REGION Network 1: Block description — Sections 1 to 3
   // ▀▀▀▀▀▀▀▀▀▀▀▀▀▀▀▀▀▀▀▀▀▀▀▀▀▀▀▀▀▀▀▀▀▀▀▀▀▀▀▀▀▀▀▀
   // 
   // TITLE:    STANDARD SYSTEM GLOBAL DATA
   // 
   // ▄▄▄▄▄▄▄▄▄▄▄▄▄▄▄▄▄▄▄▄▄▄▄▄▄▄▄▄▄▄▄▄▄▄▄▄▄▄▄▄▄▄▄▄
   //  
   // 
   // 
   // This is an essential system block that generates the internal logic and timing signals needed by 
   // all the other PAL software modules.
   // 
   // The block records the controller scan times and converts the Controller real time clock value 
   // to discrete integers, making the data globally available to all systems including non-Siemens 
   // equipment.
   // 
   // The block provides the following functions:
   // 
   //    •   Generates global logic signals (TRUE and FALSE)
   // 
   //    •   Generates the following scan synchronised timing pulses:
   //      50ms, 100ms, 200ms, 500ms, 1s and 2s
   // 
   //    •   Generates the following (1:1 mark/space) square wave signals:
   //      100ms, 200ms, 500ms, 1s and 2s
   // 
   //    •   Generates odd and even (alternating) cycle tick-tock signals
   // 
   //    •   Generates a first-cycle signal indicating the controller has just started
   // 
   //    •   Records the cycle time of the last, maximum and minimum controller cycles
   // 
   //    •   Reads the controller internal real time clock and converts the values to discrete 
   //      integer values containing: year, month, day, day of week, hour, minute, second 
   //      and millisecond
   // 
   // The block requires that the controller clock memory function is enabled.
   // 
   // The block must be the first non-debug block call within the main organisation block (OB 1).
   // 
   // 
   // 
   // 
   // 
   // ▄▄▄▄▄▄▄▄▄▄▄▄▄▄▄▄▄▄▄▄▄▄▄▄▄▄▄▄▄▄▄▄▄▄▄▄▄▄▄▄▄▄▄▄
   // 1.     BLOCK TECHNICAL SUMMARY
   // 
   // 
   //  ――――――――――――――――――――――――――――――――――――――――――
   //  NOMENCLATURE & ADDRESSING
   //  ――――――――――――――――――――――――――――――――――――――――――
   //  BLOCK TITLE         Standard System Global Data
   //  BLOCK FUNCTION GROUP    System
   //  BLOCK ADDRESS       FC 01001
   //  BLOCK SYMBOL        FC01001_StdSysGlobalData
   //  BLOCK USER ID         StdSysGlobalData
   // 
   //  ――――――――――――――――――――――――――――――――――――――――――
   //  BLOCK TYPE & USAGE
   //  ――――――――――――――――――――――――――――――――――――――――――
   //  BLOCK TYPE         Function (FC)
   //  BLOCK NUMBER        01001
   //  LANGUAGE           LAD
   //  OPTIMISED ACCESS     Yes
   //  PAL USAGE TYPE       Standard block
   // 
   //  ――――――――――――――――――――――――――――――――――――――――――
   //  METRICS
   //  ――――――――――――――――――――――――――――――――――――――――――
   //  LANGUAGE           LAD
   //  EXECUTION TIME       240.20 μs¹
   //  LOAD MEMORY         43.40 kB  (44440 bytes)
   //  WORK MEMORY             1.29 kB    (1322 bytes)
   //  ――――――――――――――――――――――――――――――――――――――――――
   //                ¹ Measured on: CPU-1515-2PN (order no. 6ES7 512-2AM02-0AB0)
   // 
   //                ━━━   ⬙⬙⬙⬙⬙⬙   ━━━
   // 
   // 
   // 
   // ▄▄▄▄▄▄▄▄▄▄▄▄▄▄▄▄▄▄▄▄▄▄▄▄▄▄▄▄▄▄▄▄▄▄▄▄▄▄▄▄▄▄▄▄
   // 2.     FUNCTIONAL DESCRIPTION
   // 
   // 
   // FC 01001 is the Standard System Global Data block, it is responsible for generating the 
   // standard set of global system signals that are common to, and used by, all other blocks within 
   // the PAL.
   // 
   // The block is one of the few essential blocks required by the PAL and it must the first block call 
   // within the main cyclic organisation block (OB 1) — it must be called before all other PAL software 
   // modules (excepting any start-of-cycle debug module — such modules will not be present in the 
   // released software)
   // 
   // The block is used to generate all the necessary logic and timing signals that are common to all
   // other PAL software modules. These signals are stored within DB21001_Dy_SysGlobalData as the 
   // data point SysSignals with UDT type UT21000_Dy_SysSignals. These signals are passed to all 
   // standard block as the parameter SYS_SIGNALS, this allows all standard blocks to access the 
   // logic and timing data parametrically¹  in accordance with IEC guidelines.
   // 
   // The block generates a second copy of the timing and logic signals and stores these as memory 
   // bit tags, these are available for use within the application blocks, these blocks are project 
   // specific (rather than the standard library blocks) and as such can directly access data points 
   // without contravening the IEC requirements. These tags are in two bytes of bit memory and form 
   // the basis of the PAL system tag table (PAL_SystemTags).
   // 
   // ――――――――――
   // ¹         The IEC guidelines state that standard (library) blocks should not directly access data 
   //      points within the controller (direct access), to do so, means that the block cannot 
   //      be a true library module that can be used on any system, it requires that system to 
   //      have an underlying set of variables that existed outside the block.
   // 
   //      The preference is for all standard (library) blocks to receive all the data they need 
   //      via parameters passed to the block (parametric access). Hence the use here of UDT 
   //      data that can be passed as a single parameter into every standard block.
   // ――――――――――
   // 
   // FC 01001 is called cyclically and monitors the cycle time of the central processor unit (CPU). The 
   // block records various cycle times: the cycle time of the previous cycle, the maximum cycle time 
   // experienced since the CPU was started and the minimum cycle time since the CPU was started. 
   // 
   // The block also decodes the CPU real time clock (RTC) value, converting it from a date_time 
   // data type to discrete integers, these being generally more accessible and easier to understand. 
   // The conversion to integers also provides simplified data for block that do not need the whole data 
   // and time information provided by the RTC, some blocks may require only time of day, or the day 
   // of the week for example. Others may only be monitoring the seconds count. It means that other 
   // blocks do not need to decode the RTC data individually.
   // 
   // All the cycle and RTC data is stored in part of the globally accessible system data block 
   // DB21001_Dy_SysGlobalData in the variable SysData, this also is a UDT (UT21001_Dy_SysData).
   // 
   // The CPU clock memory byte is used by the block (passed as a parameter) and the clock memory 
   // must be enabled in the CPU settings.
   // 
   //                ━━━   ⬙⬙⬙⬙⬙⬙   ━━━
   // 
   // 
   // 
   // ▄▄▄▄▄▄▄▄▄▄▄▄▄▄▄▄▄▄▄▄▄▄▄▄▄▄▄▄▄▄▄▄▄▄▄▄▄▄▄▄▄▄▄▄
   // 3.     DETAILED BLOCK DESCRIPTION
   // 
   // 
   // The functions of this block are broadly:
   // 
   //    1.  Generate the global logic signals
   // 
   //    2.  Generate various timing pulses and square wave signals
   // 
   //    3.  Generate cyclically dependent signals
   // 
   //    4.  Monitor and record various cycle times and properties
   // 
   //    5.  Decode the CPU real time clock and store as integer values
   // 
   // Each of these is examined in the following sections.
   // 
   // To operate correctly, the block requires the CPU clock memory to be enabled and for the specified 
   // clock memory byte to be passed as a parameter into the block. Additionally, the PAL system 
   // tag table (PAL_SystemTags) must be configured and populated with the correct mnemonic 
   // signal names. These requirements are discussed in the following sections.
   // 
   // 
   // 
   // ▂▂▂▂▂▂▂▂▂▂▂▂▂▂▂▂▂▂▂▂▂▂▂▂▂▂▂▂▂▂▂▂▂▂▂▂▂▂▂▂▂▂▂▂
   // 3.1     Enabling the clock memory byte
   // 
   // 
   // The clock memory is a CPU property that must be enabled.
   // 
   // The CPU properties are accessed from the device configuration entry in the TIA Portal project tree.
   // 
   // In the project tree select DEVICE CONFIGURATION, this opens an image of the Controller rack in 
   // the central area, right click the CPU and from the dropdown menu select PROPERTIES, this 
   // opens the property settings window in the centre-bottom area.
   // 
   // In the property settings window, under the GENERAL tab, select the SYSTEM AND CLOCK MEMORY 
   // option.
   // 
   // To enable the clock memory ensure that the ENABLE THE USE OF CLOCK MEMORY BYTE box is 
   // ticked.
   // 
   // The PAL requires that the clock byte uses byte 10 of the internal memory bits (MB10); to do this 
   // set the ADDRESS OF THE CLOCK MEMORY BYTE (MBx) to 10.
   // 
   // Note:    The section immediately above the clock memory bits, SYSTEM MEMORY BITS, 
   //      must not be enabled, ensure that the ENABLE USE OF SYSTEM MEMORY BYTE box 
   //      is unticked.
   // 
   // 
   // 
   // ▂▂▂▂▂▂▂▂▂▂▂▂▂▂▂▂▂▂▂▂▂▂▂▂▂▂▂▂▂▂▂▂▂▂▂▂▂▂▂▂▂▂▂▂
   // 3.2     The PAL System signals (logic and timing)
   // 
   // 
   // The PAL system signals (logic and timing signals) are stored in two formats, first as a UDT data 
   // structure (UT21000_Dy_SysSignals) in the system global data block (DB21001_Dy_SysGlobalData) 
   // in the variable SysSignals. This form of the system signals is designed to be passed as a 
   // parameter to all standard (library) modules.
   // 
   // Secondly, the same data is stored in bit memories, these can be accessed globally in all 
   // application (project specific) blocks. The bit memories used to store the system signals are MB0 
   // and MB1; the individual signals within the bytes being given symbolic tags in the tag table 
   // PAL_SystemTags.
   // 
   // Both forms of the data are discussed further in the following sections:
   // 
   // Note:    There is absolutely no difference between the two form of the signals, it is simply a 
   //      question of which to use under what circumstances: parametric for library modules, 
   //      direct for application modules.
   // 
   // 
   // 
   // ▁▁▁▁▁▁▁▁▁▁▁▁▁▁▁▁▁▁▁▁▁▁▁▁▁▁▁▁▁▁▁▁▁▁▁▁▁▁▁▁▁▁▁▁
   // 3.2.1     System signals: parametric access and direct access
   // 
   // 
   // The IEC guidelines state that standard (library) blocks should not directly access data points 
   // within the controller (direct access), to do so, means that the block cannot be a true library 
   // module that can be used on any system, it requires that system to have an under-lying set of 
   // variables that existed outside the block.
   // 
   // The preference is for all standard (library) block to receive all the data they need via parameters 
   // passed to the block (parametric access). Hence the use here of UDT data that can be passed as
   // a single parameter into every standard block.
   // 
   // The application blocks are by their nature, specific to the project being developed, they are not 
   // library modules. As such the application modules can use direct access to read the system 
   // signals. 
   // 
   // Hence the two versions:
   // 
   //    •   Parametric access — UDT parameter for standard modules
   //    •   Direct access — memory bits for application modules
   // 
   // Examining these in turn:
   // 
   // 
   // 
   // ▁▁▁▁▁▁▁▁▁▁▁▁▁▁▁▁▁▁▁▁▁▁▁▁▁▁▁▁▁▁▁▁▁▁▁▁▁▁▁▁▁▁▁▁
   // 3.2.2     UDT system signals for parametric access
   // 
   // 
   // The system logic and timing signals for parametric access are stored in 
   // DB21001_Dy_SysGlobalData in the variable SysSignals; this variable is a UDT of type 
   // UT21000_Dy_SysSignals, it contains the 16 logic and timing signals shown below:
   // 
   //  UT21000_Dy_SysGlobalData
   //  ――――――――――――――――――――――――――――――――――――――――――
   //  SIGNAL NAME          FUNCTION                     TYPE
   //  ――――――――――――――――――――――――――――――――――――――――――
   //  _False              System Logic   — Always FALSE            Bool
   //  _True             System Logic   — Always TRUE              Bool
   //  _50ms             System Timing — 50 ms pulse           Bool
   //  _100ms              System Timing — 100 ms pulse            Bool 
   //  _200ms              System Timing — 200 ms pulse            Bool 
   //  _500ms              System Timing — 500 ms pulse            Bool 
   //  _1s             System Timing — 1 s pulse              Bool 
   //  _2s             System Timing — 2 s pulse              Bool 
   //  _CycleTick             System Timing — Cycle tick (odd cycles)         Bool
   //  _CycleTock            System Timing — Cycle tock (even cycle)        Bool
   //  _CycleFirst            System Timing — First cycle detected           Bool
   //  _100msSqW         System Timing — 100 ms square wave        Bool 
   //  _200msSqW         System Timing — 200 ms square wave        Bool 
   //  _500msSqW         System Timing — 500 ms square wave        Bool 
   //  _1sSqW              System Timing — 1 s square wave             Bool
   //  _2sSqW              System Timing — 2 s square wave             Bool 
   //  ――――――――――――――――――――――――――――――――――――――――――
   // 
   // 
   // This data is passed as a parameter to all standard (library) blocks; the parameter is named 
   // SYS_SIGNALS on all standard blocks, and is always the first IN parameter:
   // 
   // 
   //                        ┌─────────────
   //  ──────────────────────┤ FCxxxxx_StdBlock
   //                        ├───────────
   //      "DB21001_DY_StdGlobalData".SysSignals ─┤ SYS_SIGNALS
   //                        │
   //                        │
   // 
   // 
   // 
   // ▁▁▁▁▁▁▁▁▁▁▁▁▁▁▁▁▁▁▁▁▁▁▁▁▁▁▁▁▁▁▁▁▁▁▁▁▁▁▁▁▁▁▁▁
   // 3.2.3     Bit memory direct access and the PAL system tag table
   // 
   // 
   // The clock memory signals generated by the CPU (stored in MB10) and all the global logic and 
   // timing signals generated by this block (stored in MB0 and MB1, see Table 3.1) are given 
   // symbolic names (tags) that are then used throughout the remaining PAL software modules.
   // 
   // Note:    It is unusual for data to be stored in bit memories; the PAL generally uses data 
   //      blocks to store information. 
   // 
   //      An exception is made for the clock memory (this has to be stored in bit memories) 
   //      and for the global logic and timing signals. These are used frequently within software 
   //      modules and allocating the signals to memory bits means that the tags are shorter 
   //      and more easily recognised a system signals. It is also quicker to enter these signals.
   // 
   // The tags for these three bytes (MB0, MB1 and MB10) are specified in the PLC TAGS entry in the 
   // project tree, and are stored in the tag table: 
   // 
   //      PAL_SystemTags
   // 
   // This tag table is provided as standard as part of the PAL. A full list of its contents is provided 
   // in the table below.
   // 
   // The PAL_SystemTags tag table is a fixed tag table and is a fundamental part of the PAL. 
   // IT MUST NOT BE MODIFIED. 
   // 
   // The bit memories contained in the bytes MB0, MB1 and MB10 are similarly reserved by the PAL 
   // and must these not be reallocated, renamed or used in any other tag table.
   // 
   // The memory bit system signals are given identical names to those in the 
   // UT21000_Dy_SysSignals data type (those used for parametric access, see § 3.2.2); as follows:
   // 
   // 
   //  ――――――――――――――――――――――――――――――――――――――――――
   //  NAME          TYPE  ADDRESS DESCRIPTION
   //  ――――――――――――――――――――――――――――――――――――――――――
   //  _SysSignals        Int      %MW0   System signals — Logic and timing
   //  _SysSignals01         Byte   %MB0    System mem byte 01 — Logic and timing
   //  _False            Bool     %M0.0   System Logic — Always FALSE
   //  _True           Bool     %M0.1   System Logic — Always TRUE
   //  _50ms           Bool     %M0.2   System Timing — 50 ms pulse 
   //  _100ms            Bool     %M0.3   System Timing — 100 ms pulse 
   //  _200ms            Bool     %M0.4   System Timing — 200 ms pulse 
   //  _500ms            Bool     %M0.5   System Timing — 500 ms pulse 
   //  _1s           Bool     %M0.6   System Timing — 1 s pulse 
   //  _2s           Bool     %M0.7   System Timing — 2 s pulse 
   //  ――――――――――――――――――――――――――――――――――――――――――
   //  _SysSignals02         Byte   %MB1    System mem byte 02 — cycle & square wave
   //  _CycleTick           Bool     %M1.0   System Timing — Cycle tick (odd cycles)
   //  _CycleTock          Bool     %M1.1   System Timing — Cycle tock (even cycle)
   //  _CycleFirst          Bool     %M1.2   System Timing — First cycle detected
   //  _100msSqW       Bool     %M1.3   System Timing — 100 ms square wave 
   //  _200msSqW       Bool     %M1.4   System Timing — 200 ms square wave 
   //  _500msSqW       Bool     %M1.5   System Timing — 500 ms square wave 
   //  _1sSqW            Bool     %M1.6   System Timing — 1 s square wave 
   //  _2sSqW            Bool     %M1.7   System Timing — 2 s square wave 
   //  ――――――――――――――――――――――――――――――――――――――――――
   //  _ClockMem         Byte   %MB10     Clock Memory (populated by the CPU)
   //  _ClockMem_100msSqW    Bool     %M10.0    Clock Memory — 10.0 Hz square wave
   //  _ClockMem_200msSqW    Bool     %M10.1    Clock Memory — 5.00 Hz square wave
   //  _ClockMem_400msSqW    Bool     %M10.2    Clock Memory — 2.50 Hz square wave
   //  _ClockMem_500msSqW    Bool     %M10.3    Clock Memory — 2.00 Hz square wave
   //  _ClockMem_800msSqW    Bool     %M10.4    Clock Memory — 1.25 Hz square wave
   //  _ClockMem_1000msSqW  Bool     %M10.5    Clock Memory — 1.00 Hz square wave
   //  _ClockMem_1600msSqW  Bool     %M10.6    Clock Memory — 0.62 Hz square wave
   //  _ClockMem_2000msSqW  Bool     %M10.7    Clock Memory — 0.50 Hz square wave
   //  ――――――――――――――――――――――――――――――――――――――――――
   // 
   // 
   // All PAL system tags contained within the PAL_SystemTags tag table are identified by a leading 
   // underscore character (_).
   // 
   // The PAL system tags are named according to the following conventions:
   // 
   //    1.  Each tag is prefixed with the underscore [ _ ] character
   // 
   //    2.  The remaining tag name is written in camel case 
   // 
   //    3.  The name (including prefix) must be no more than 24 characters 
   // 
   //    4.  It is permissible to separate parts of the name with an underscore [ _ ] character 
   //      (e.g. _ClockMem_100msSqW)
   // 
   //    5.  Units (such as milliseconds, ms) are not capitalised
   // 
   //    6.  The dash/hyphen [-] is not to be used (use the underscore in-stead)
   // 
   //    7.  Only use the characters [a-z], [A-Z], the numbers [0-9], and the underscore [ _ ]
   // 
   // All PAL system tags have a brief explanation of what the tag does stored in the comment field 
   // of the tag.
   // 
   // 
   // 
   // ▂▂▂▂▂▂▂▂▂▂▂▂▂▂▂▂▂▂▂▂▂▂▂▂▂▂▂▂▂▂▂▂▂▂▂▂▂▂▂▂▂▂▂▂
   // 3.3     General point for the following sections
   // 
   // 
   // The following sections refer to the logic and timing signals generated by the block. These can 
   // refer to either the parametric version of the data stored as a UDT or the direct access version 
   // stored as memory bits. The name of each signal is the same in either case (e.g. _True, _False &c.); 
   // the difference is that the parametric version will be proceeded by the SYS_SIGNALS parameter 
   // name e.g.:
   //           #SYS_SIGNALS._True
   // 
   // For brevity, the following section just refer to the signal name e.g. _True; where the parametric 
   // access is used, this should be preceded by #SYS_SIGNALS.
   // 
   // 
   // 
   // ▂▂▂▂▂▂▂▂▂▂▂▂▂▂▂▂▂▂▂▂▂▂▂▂▂▂▂▂▂▂▂▂▂▂▂▂▂▂▂▂▂▂▂▂
   // 3.4     Global logic signals
   // 
   // 
   // The block generates two fixed logic signals, these are allocated as follows:
   // 
   // 
   //  ――――――――――――――――――――――――――――――――――――――――――
   //  NAME          TYPE  DESCRIPTION
   //  ――――――――――――――――――――――――――――――――――――――――――
   //  _False            Bool     System Logic Bit — Always FALSE
   //  _True           Bool     System Logic Bit — Always TRUE
   //  ――――――――――――――――――――――――――――――――――――――――――
   // 
   // 
   // The two signals _False and _True are logically testable signals, the _False signal being always 
   // set to 0 and the _True signal being always set to 1.
   // 
   // These two signals should be considered read only; other software modules must not change the 
   // state of these signals.
   // 
   // This block, FC 01001, will ensure that the _False signal is always set to 0 and the _True signal is 
   // always set to 1.
   // 
   // 
   // 
   // ▂▂▂▂▂▂▂▂▂▂▂▂▂▂▂▂▂▂▂▂▂▂▂▂▂▂▂▂▂▂▂▂▂▂▂▂▂▂▂▂▂▂▂▂
   // 3.5     Global timing signals
   // 
   // 
   // The block generates two types of timing signals: scan synchronised pulses that are active for a 
   // single controller cycle (scan) and scan synchronised even mark/space ratio square waves.
   // 
   // Both types of timing signal are derived from the CPU clock memory functions (see table below). 
   // Within the PAL the clock memory is given the tag _ClockMem and is assigned to memory 
   // byte MB10. The CPU populates the _ClockMem byte with eight square wave signals each with a 
   // different frequency.
   // 
   // 
   //  ――――――――――――――――――――――――――――――――――――――――――
   //  NAME          TYPE  ADDRESS DESCRIPTION
   //  ――――――――――――――――――――――――――――――――――――――――――
   //  _ClockMem         Byte   %MB10     Clock Memory (populated by the CPU)
   //  _ClockMem_100msSqW    Bool     %M10.0    Clock Memory — 10.0 Hz square wave
   //  _ClockMem_200msSqW    Bool     %M10.1    Clock Memory — 5.00 Hz square wave
   //  _ClockMem_400msSqW    Bool     %M10.2    Clock Memory — 2.50 Hz square wave
   //  _ClockMem_500msSqW    Bool     %M10.3    Clock Memory — 2.00 Hz square wave
   //  _ClockMem_800msSqW    Bool     %M10.4    Clock Memory — 1.25 Hz square wave
   //  _ClockMem_1000msSqW  Bool     %M10.5    Clock Memory — 1.00 Hz square wave
   //  _ClockMem_1600msSqW  Bool     %M10.6    Clock Memory — 0.62 Hz square wave
   //  _ClockMem_2000msSqW  Bool     %M10.7    Clock Memory — 0.50 Hz square wave
   //  ――――――――――――――――――――――――――――――――――――――――――
   // 
   // 
   // Each of these square wave signals is free running (they run independently to the CPU cycle), 
   // but are synchronised with each other (i.e. they all start at the same time and have rising edges 
   // that coincide with each other in multiples of 100 ms).
   // 
   // This block uses the CPU clock memory signals to generate the derived scan synchronised timing 
   // pulses and square waves.
   // 
   // Examining these in turn:
   // 
   // 
   // 
   // ▁▁▁▁▁▁▁▁▁▁▁▁▁▁▁▁▁▁▁▁▁▁▁▁▁▁▁▁▁▁▁▁▁▁▁▁▁▁▁▁▁▁▁▁
   // 3.5.1     Scan synchronised timing pulses
   // 
   // 
   // This block produces six individual timing pulses:
   // 
   // 
   //  ――――――――――――――――――――――――――――――――――――――――――
   //  NAME          TYPE  DESCRIPTION
   //  ――――――――――――――――――――――――――――――――――――――――――
   //  _50ms           Bool     System Timing — 50 ms pulse 
   //  _100ms            Bool     System Timing — 100 ms pulse 
   //  _200ms            Bool     System Timing — 200 ms pulse 
   //  _500ms            Bool     System Timing — 500 ms pulse 
   //  _1s           Bool     System Timing — 1 s pulse 
   //  _2s           Bool     System Timing — 2 s pulse 
   //  ――――――――――――――――――――――――――――――――――――――――――
   // 
   // 
   // Each pulse is active for a single CPU cycle, and is activated at the start of the cycle following the 
   // rising edge of the associated _ClockMem bit (there is an exception for the _50ms pulse; this is 
   // explained at the end of this section).
   // 
   // The _ClockMem signals are free running square wave signals that are completely independent 
   // of the CPU cycle times, this means that the signal can change state partway through a controller 
   // cycle, if each block within the controller were evaluating the clock memory for timing 
   // arrangements, it would mean that some blocks would see the timing signal in one state (before 
   // it changed) and others would see it in the second state (after it changed) and this can lead to 
   // inconsistences with software reactions.
   // 
   // This type of reaction (signals that are independent of the controller cycle) is referred to as 
   // asynchronous behaviour and it is generally to be avoided.
   // 
   // To avoid this problem, this block (FC 01001) monitors the clock memory signals, if the block 
   // detects a rising edge on any of the clock memory signals (the edge may have occurred in the 
   // preceding cycle, but will not be detected until the block is executed at the start of the following 
   // cycle), it activates the associated timing pulse, the timing pulse is then deactivated the next 
   // time FC 01001 is called.
   // 
   // FC 01001 is called as the first executable block in the main organisation block (OB 1), thus 
   // any timing pulses are effectively present to all the other blocks for the cycle within which it is 
   // triggered. This is called scan synchronisation.
   // 
   // 
   // 
   // ▁▁▁▁▁▁▁▁▁▁▁▁▁▁▁▁▁▁▁▁▁▁▁▁▁▁▁▁▁▁▁▁▁▁▁▁▁▁▁▁▁▁▁▁
   // Scan synchronised timing pulse accuracy
   // 
   // 
   // The accuracy of the timing pulse is compromised by the scan synchronisation actions of 
   // FC 01001. 
   // 
   // If for example, the 100 ms clock memory square wave went to high state just after FC 01001 
   // had been executed in cycle n, it would not be detected until FC 01001 was executed in 
   // cycle n + 1. If in this example the cycle is approximately 12 ms, the timing pulse would be 
   // delayed by 12 ms.
   // 
   // Thus the maximum inaccuracy of the timing pulse is limited to the cycle time of the controller.
   // 
   // These inaccuracies are not cumulative. The delay of up to one cycle is applicable to each pulse in 
   // turn; the pulse will always be activated no later than one cycle duration from the time at which 
   // the clock memory signal goes high.
   // 
   // 
   // 
   // ▁▁▁▁▁▁▁▁▁▁▁▁▁▁▁▁▁▁▁▁▁▁▁▁▁▁▁▁▁▁▁▁▁▁▁▁▁▁▁▁▁▁▁▁
   // Generating the 50 ms timing pulse
   // 
   // 
   // Each of the timing pulse signals: _100ms, _200ms, _500ms, _1s and _2s are generated by 
   // detecting a rising edge on each of the corresponding clock memory signals: 
   // _ClockMem_100msSqW, _ClockMem_200msSqW, _ClockMem_500msSqW, 
   // _ClockMem_1000msSqW and _ClockMem_2000msSqW. 
   // 
   // There is no 50 ms square wave provided by the clock memory function; to generate the 50 ms 
   // timing pulse, the pulse is generated on both the rising and falling edge of the 100 ms clock 
   // memory square wave.
   // 
   // The clock memory square wave have an equal mark/space ratio, thus the falling edge occurs 
   // after 50 ms.
   // 
   // 
   // 
   // ▁▁▁▁▁▁▁▁▁▁▁▁▁▁▁▁▁▁▁▁▁▁▁▁▁▁▁▁▁▁▁▁▁▁▁▁▁▁▁▁▁▁▁▁
   // 3.5.2     Scan synchronised timing square waves
   // 
   // 
   // This block produces five individual timing square wave signals:
   // 
   // 
   //  ――――――――――――――――――――――――――――――――――――――――――
   //  NAME          TYPE  DESCRIPTION
   //  ――――――――――――――――――――――――――――――――――――――――――
   //  _100msSqW       Bool     System Timing — 100 ms square wave 
   //  _200msSqW       Bool     System Timing — 200 ms square wave 
   //  _500msSqW       Bool     System Timing — 500 ms square wave 
   //  _1sSqW            Bool     System Timing — 1 s square wave 
   //  _2sSqW            Bool     System Timing — 2 s square wave 
   //  ――――――――――――――――――――――――――――――――――――――――――
   // 
   // 
   // These signals are again scan synchronised in a similar manner to the timing pulses, the 
   // rising and falling edges of the scan synchronised timing square wave occur at the start of the 
   // cycle following the change in state of the clock memory square wave.
   // 
   // 
   // 
   // ▁▁▁▁▁▁▁▁▁▁▁▁▁▁▁▁▁▁▁▁▁▁▁▁▁▁▁▁▁▁▁▁▁▁▁▁▁▁▁▁▁▁▁▁
   // Scan synchronised timing square wave accuracy
   // 
   // Again, the scan synchronisation actions of FC 01001 compromise the accuracy of the timing 
   // square wave signals and again by the same amount, each rising and falling edge of the square 
   // wave can be delayed by up to the duration of one cycle.
   // 
   // These inaccuracies are again, not cumulative. The period of the square wave (rising edge to 
   // rising edge) will be no more than the duration of a single cycle for each square wave cycle.
   // 
   // The mark/space ratio of the timing square wave will also be compromised, again by up to one 
   // cycle duration.
   // 
   // 
   // 
   // ▂▂▂▂▂▂▂▂▂▂▂▂▂▂▂▂▂▂▂▂▂▂▂▂▂▂▂▂▂▂▂▂▂▂▂▂▂▂▂▂▂▂▂▂
   // 3.6     Cyclically dependent signals
   // 
   // 
   // The block generates three cycle dependent signals:
   // 
   // 
   //  ――――――――――――――――――――――――――――――――――――――――――
   //  NAME          TYPE  DESCRIPTION
   //  ――――――――――――――――――――――――――――――――――――――――――
   //  _CycleTick           Bool     System Timing — Cycle tick (odd cycles)
   //  _CycleTock          Bool     System Timing — Cycle tock (even cycle)
   //  _CycleFirst          Bool     System Timing — First cycle detected
   //  ――――――――――――――――――――――――――――――――――――――――――
   // 
   // 
   // The first two of these signals (_CycleTick and _CycleTock) are alternating signals that change 
   // state at the start of each cycle, the _CycleTick being active on every odd cycle since the CPU 
   // Started (cycles 1, 3, 5, 7 …).
   // 
   // _CycleTock activates on each even numbered cycle since the CPU started (cycles 2, 4, 6, 8 …).
   // 
   // The _CycleTick and _CycleTock signals are often used as “dead-man” signals that show the CPU 
   // is running.
   // 
   // The _CycleFirst signal is active on the first cycle of the CPU after a STOP → RUN transition.
   // 
   // The _CycleFirst signal is an important signal and is generally used to set the controller to a given 
   // condition. It should be interpreted as telling the software that the processor has just started and 
   // all modules should be initialised and set to the correct start-up conditions.
   // 
   // The _CycleFirst signal is generated by using the system start information block (RD_SINFO), this 
   // is called with the system data structure SI_ProgramCycle, see § 9.
   // 
   // 
   // 
   // ▁▁▁▁▁▁▁▁▁▁▁▁▁▁▁▁▁▁▁▁▁▁▁▁▁▁▁▁▁▁▁▁▁▁▁▁▁▁▁▁▁▁▁▁
   // 3.6.1     Record various cycle times and properties
   // 
   // 
   // The block reads various cycle time values and generates a cycle count that is incremented at 
   // the start of each cycle.
   // 
   // This data is stored in the system data block: DB21001_Dy_SysGlobalData in the variable 
   // SysData. The storage location is passed to the block as a parameter (SYS_DATA) of data type 
   // UT21001_Dy_SysData (see Section 5 for details of the full structure).
   // 
   // The following data is recorded:
   // 
   // 
   //  UT21001_Dy_SysGlobalData (Partial contents)
   //  ――――――――――――――――――――――――――――――――――――――――――
   //  SIGNAL NAME          FUNCTION                     TYPE
   //  ――――――――――――――――――――――――――――――――――――――――――
   //  CycTime_Prev          Previous cycle time (ms)             Real
   //  CycTime_Max          Maximum cycle time - since start-up (ms)       Real
   //  CycTime_Min        Minimum cycle time - since start-up (ms)        Real
   //  Cyc_Counter         Cycle rolling counter - incremented each scan     UDint
   //  ――――――――――――――――――――――――――――――――――――――――――
   // 
   // 
   // The data for the min, max and previous cycle times is provided by the system function RT_INFO, 
   // this returns the various cycle times in LTime data format, this is converted to a real number that 
   // specifies the cycle times in milliseconds.
   // 
   // For example if the signal CycTime_Prev returned a value of 15.36, it would indicate that the 
   // duration of the previous cycle was 15.36 ms.
   // 
   // The Cyc_Counter signal is simply an unsigned double integer (UDint) that is incremented by one 
   // each scan. This is done within FC 01001, the counter can count up to 4.3 billion cycles 
   // (4,294,967,296) before repeating (at an average cycle time of 15 ms, it would be two years 
   // before the counter wrapped around and started again at zero).
   // 
   // The Cyc_Counter signal is reset to zero if the CPU is restarted (_CycleFirst signal is triggered), it is 
   // also reset to zero if the count exceeds the maximum value for a UDint (4,294,967,296).
   // 
   // 
   // 
   // ▂▂▂▂▂▂▂▂▂▂▂▂▂▂▂▂▂▂▂▂▂▂▂▂▂▂▂▂▂▂▂▂▂▂▂▂▂▂▂▂▂▂▂▂
   // 3.7     Real time clock (RTC) data
   // 
   // 
   // The CPU maintains an internal real time clock (RTC), this is generally synchronised to an external 
   // time server (a SCADA system for example). The RTC contains date, time and day of week 
   // information and can be accessed using the system function RD_LOC_T. This function returns the 
   // RTC value in a variable that uses a date and time based data type (DateTime, DTL, LDT &c.).
   // 
   // The DTL data type is used by preference, it is a structured data type, with fields for each time and 
   // date component, it allows each field to be easily split out and stored separately. It does, 
   // however, theoretically provide accuracy down to the nanosecond, in practice, most of the 
   // nanosecond digits are set to zero with only the three most significant digits being populated. 
   // 
   // Essentially it just gives an accuracy of milliseconds, and it is this millisecond value that is stored.
   // 
   // FC 01001 converts the RTC data to a series of unsigned integers that are stored as part of the 
   // UT21001_Dy_SysGlobalData data type that is passed to the block as the parameter 
   // (SYSTEM_DATA). It provides the following information:
   // 
   // Note:    The RTC data is local to the time zone set in the CPU and adopts any local daylight 
   //      saving that is in effect.
   // 
   // 
   //  UT21001_Dy_SysGlobalData (partial contents)
   //  ――――――――――――――――――――――――――――――――――――――――――
   //  SIGNAL NAME          FUNCTION                     TYPE
   //  ――――――――――――――――――――――――――――――――――――――――――
   //  RTC_Year            Year (returns a value in the range 1970 to 2262)     UInt
   //  RTC_Month         Month (1-12 representing Jan to Dec)        UInt
   //  RTC_Day          Day of month (1-31)                  UInt
   //  RTC_DayOfWeek         Day of week (1-7, where 1=Sunday, 7=Saturday)    UInt
   //  RTC_Hour           Hour of day (0-23)                UInt
   //  RTC_Minute           Minutes (0-59)                   UInt
   //  RTC_Second         Seconds (0-59)                  UInt
   //  RTC_Millisecond         Milliseconds (0-999)                  UInt
   //  ――――――――――――――――――――――――――――――――――――――――――
   // 
   //                ━━━   ⬙⬙⬙⬙⬙⬙   ━━━
END_REGION

REGION Network 2: Block description — Sections 4 to 11
   // ▄▄▄▄▄▄▄▄▄▄▄▄▄▄▄▄▄▄▄▄▄▄▄▄▄▄▄▄▄▄▄▄▄▄▄▄▄▄▄▄▄▄▄▄
   // 4.     PARAMETERS
   // 
   // 
   // The following parameters are associated with the block:
   // 
   //  
   //  ――――――――――――――――――――――――――――――――――――――――――
   //  PARAM         FUNCTION                    TYPE      IN-OUT 
   //  ――――――――――――――――――――――――――――――――――――――――――
   //  CLOCK_MEM     The clock memory byte (within the PAL this      Byte      In
   //           is always MB10)
   // 
   //  SYS_SIGNALS      The system logic and timing signals for       UT21000    InOut
   //           parametric access
   // 
   //  SYS_DATA      The system data storage structure interface,   UT21001    InOut
   //           holds the cycle & RTC data
   // 
   //  SYS_SIGNAL_TAGS   The system logic and timing signals for       Int      Out
   //           direct access
   //  ――――――――――――――――――――――――――――――――――――――――――
   // 
   //                ━━━   ⬙⬙⬙⬙⬙⬙   ━━━
   // 
   // 
   // 
   // ▄▄▄▄▄▄▄▄▄▄▄▄▄▄▄▄▄▄▄▄▄▄▄▄▄▄▄▄▄▄▄▄▄▄▄▄▄▄▄▄▄▄▄▄
   // 5.     DATA STRUCTURES AND USAGE (AND INSTANCE DATA BLOCKS)
   // 
   // 
   // The block has the following associated data structure:
   // 
   // 
   //  ――――――――――――――――――――――――――――――――――――――――――
   //  DATA STRUCTURE             DESCRIPTION
   //  ――――――――――――――――――――――――――――――――――――――――――
   //  UT01000_St_SysRevision          Revision information for this block
   //  UT01001_St_SysLicence           Licence information for this block
   //  UT21000_Dy_SysSignals           System signals (logic and timing) storage structure
   //  UT21001_Dy_SysData          System data storage structure
   //  ――――――――――――――――――――――――――――――――――――――――――
   // 
   // 
   // 
   // ▂▂▂▂▂▂▂▂▂▂▂▂▂▂▂▂▂▂▂▂▂▂▂▂▂▂▂▂▂▂▂▂▂▂▂▂▂▂▂▂▂▂▂▂
   // 5.1     UT01000_St_SysRevision
   // 
   // 
   // Used to store the revision information for the block:
   // 
   // 
   //  UT01000_St_SysRevision    (full contents)
   //  ――――――――――――――――――――――――――――――――――――――――――
   //  SIGNAL NAME          FUNCTION                     TYPE
   //  ――――――――――――――――――――――――――――――――――――――――――
   //  REV_BLOCK          Block number (of this block)             String[7]
   //  REV_NUMBER          Revision status and revision number (for this block)   String[20]
   //  REV_DATE          Revision date in format YYYY-MM-DD          String[10]
   //  REV_AUTHOR        Revision author (initial and surname)        String[20]
   //  ――――――――――――――――――――――――――――――――――――――――――
   // 
   // 
   // 
   // ▂▂▂▂▂▂▂▂▂▂▂▂▂▂▂▂▂▂▂▂▂▂▂▂▂▂▂▂▂▂▂▂▂▂▂▂▂▂▂▂▂▂▂▂
   // 5.2     UT01001_St_SysLicence
   // 
   // 
   // Used to store the licencing information for the block:
   // 
   // 
   //  UT01001_St_SysLicence    (full contents)
   //  ――――――――――――――――――――――――――――――――――――――――――
   //  SIGNAL NAME          FUNCTION                     TYPE
   //  ――――――――――――――――――――――――――――――――――――――――――
   //  LICENCE_TYPE         Type of licence under which the block can be used  String[20]
   //  COPYRIGHT           Copyright holder of the software           String[30]
   //  ――――――――――――――――――――――――――――――――――――――――――
   // 
   // 
   // 
   // ▂▂▂▂▂▂▂▂▂▂▂▂▂▂▂▂▂▂▂▂▂▂▂▂▂▂▂▂▂▂▂▂▂▂▂▂▂▂▂▂▂▂▂▂
   // 5.3     UT21000_Dy_SysSignals
   // 
   // 
   // Used to store system logic and timing signals for parametric access:
   // 
   // 
   //  UT21000_Dy_SysSignals (full contents)
   //  ――――――――――――――――――――――――――――――――――――――――――
   //  SIGNAL NAME          FUNCTION                     TYPE
   //  ――――――――――――――――――――――――――――――――――――――――――
   //  _False              System Logic   — Always FALSE            Bool
   //  _True             System Logic   — Always TRUE              Bool
   //  _50ms             System Timing — 50 ms pulse           Bool
   //  _100ms              System Timing — 100 ms pulse            Bool 
   //  _200ms              System Timing — 200 ms pulse            Bool 
   //  _500ms              System Timing — 500 ms pulse            Bool 
   //  _1s             System Timing — 1 s pulse              Bool 
   //  _2s             System Timing — 2 s pulse              Bool 
   //  _CycleTick             System Timing — Cycle tick (odd cycles)         Bool
   //  _CycleTock            System Timing — Cycle tock (even cycle)        Bool
   //  _CycleFirst            System Timing — First cycle detected           Bool
   //  _100msSqW         System Timing — 100 ms square wave        Bool 
   //  _200msSqW         System Timing — 200 ms square wave        Bool 
   //  _500msSqW         System Timing — 500 ms square wave        Bool 
   //  _1sSqW              System Timing — 1 s square wave             Bool
   //  _2sSqW              System Timing — 2 s square wave             Bool 
   //  ――――――――――――――――――――――――――――――――――――――――――
   // 
   // 
   // 
   // ▂▂▂▂▂▂▂▂▂▂▂▂▂▂▂▂▂▂▂▂▂▂▂▂▂▂▂▂▂▂▂▂▂▂▂▂▂▂▂▂▂▂▂▂
   // 5.4     UT21001_Dy_SysData
   // 
   // 
   // Used to store system cycle and time data:
   // 
   // 
   //  UT21001_Dy_SysData (full contents)
   //  ――――――――――――――――――――――――――――――――――――――――――
   //  SIGNAL NAME          FUNCTION                     TYPE
   //  ――――――――――――――――――――――――――――――――――――――――――
   //  CycTime_Prev          Previous cycle time (ms)             Real
   //  CycTime_Max          Maximum cycle time - since start-up (ms)       Real
   //  CycTime_Min        Minimum cycle time - since start-up (ms)        Real
   //  Cyc_Counter         Cycle rolling counter - incremented each scan     UDint
   // 
   //  RTC_Year            Year (returns a value in the range 1970 to 2262)     UInt
   //  RTC_Month         Month (1-12 representing Jan to Dec)        UInt
   //  RTC_Day          Day of month (1-31)                  UInt
   //  RTC_DayOfWeek         Day of week (1-7, where 1=Sunday, 7=Saturday)    UInt
   //  RTC_Hour           Hour of day (0-23)                UInt
   //  RTC_Minute           Minutes (0-59)                   UInt
   //  RTC_Second         Seconds (0-59)                  UInt
   //  RTC_Millisecond         Milliseconds (0-999)                  UInt
   //  ――――――――――――――――――――――――――――――――――――――――――
   // 
   // 
   //                ━━━   ⬙⬙⬙⬙⬙⬙   ━━━
   // 
   // 
   // 
   // ▄▄▄▄▄▄▄▄▄▄▄▄▄▄▄▄▄▄▄▄▄▄▄▄▄▄▄▄▄▄▄▄▄▄▄▄▄▄▄▄▄▄▄▄
   // 6.     CONSTANTS AND TEMPORARY (LOCAL) DATA
   // 
   // 
   // The following constants and temporary data storage are used:
   // 
   // 
   //  Temporary (local) data
   //  ――――――――――――――――――――――――――――――――――――――――――
   //  SIGNAL NAME          FUNCTION                  TYPE
   //  ――――――――――――――――――――――――――――――――――――――――――
   //  revInfo             Revision information for the block         UT01000
   //  licInfo           Licensing information for the block      UT01001
   //  SI_ProgramCycle       Used by RD_SINFO, holds first scan data   SI_ProgramCycle
   //  SI_StartUp         Required by RD_SINFO (not used)         SI_StartUp
   //  wrkInt           Working storage area (integer)          Int
   //  wrkDInt           Working storage area (double integer)         DInt
   //  wrkReal           Working storage area (real)             Real
   //  wrkLTime           Working storage area (long time)         LT
   //  wrkDTL            Working storage area (DateTime long)      DTL
   //  ――――――――――――――――――――――――――――――――――――――――――
   // 
   // 
   //                ━━━   ⬙⬙⬙⬙⬙⬙   ━━━
   // 
   // 
   // 
   // ▄▄▄▄▄▄▄▄▄▄▄▄▄▄▄▄▄▄▄▄▄▄▄▄▄▄▄▄▄▄▄▄▄▄▄▄▄▄▄▄▄▄▄▄
   // 7.     BLOCK CALLS
   // 
   // 
   // There are no PAL block calls from within this block.
   // 
   //                ━━━   ⬙⬙⬙⬙⬙⬙   ━━━
   // 
   // 
   // 
   // ▄▄▄▄▄▄▄▄▄▄▄▄▄▄▄▄▄▄▄▄▄▄▄▄▄▄▄▄▄▄▄▄▄▄▄▄▄▄▄▄▄▄▄▄
   // 8.     ASSOCIATED BLOCKS
   // 
   // 
   // This is a stand-alone block and is not associated with any other blocks.
   // 
   //                ━━━   ⬙⬙⬙⬙⬙⬙   ━━━
   // 
   // 
   // 
   // ▄▄▄▄▄▄▄▄▄▄▄▄▄▄▄▄▄▄▄▄▄▄▄▄▄▄▄▄▄▄▄▄▄▄▄▄▄▄▄▄▄▄▄▄
   // 9.     SYSTEM BLOCK CALLS AND SYSTEM DATA TYPES
   // 
   // 
   // The following calls are made to system blocks:
   // 
   // 
   //  System block calls
   //  ――――――――――――――――――――――――――――――――――――――――――
   //  BLOCK          TITLE             DESCRIPTION  
   //  ――――――――――――――――――――――――――――――――――――――――――
   //  RD_SINFO          Read OB start info       Used to read the OB start information
   //                            including first scan information
   // 
   //  RT_INFO             Read runtime statistics    Used to return the previous, min 
   //                            and max cycle times
   // 
   //  RD_LOC_T             Read the local RTC time    Reads the CPU real time clock 
   //  ――――――――――――――――――――――――――――――――――――――――――
   // 
   // 
   // The following system data types are required:
   // 
   // 
   //  SI_ProgramCycle (System Data Type)
   //  ――――――――――――――――――――――――――――――――――――――――――
   //  SIGNAL NAME          FUNCTION                     TYPE
   //  ――――――――――――――――――――――――――――――――――――――――――
   //  SI_Format          Start information format, indicates if the         USInt
   //               current OB is using block optimisation
   //                 16#FF = No information
   //                 16#FE = Block optimised
   // 
   //  OB_Class           Class  of the calling OB, for this data structure     USInt 
   //               the result is always 1 (indicating cyclic OB)
   // 
   //  OB_Nr           Number of the calling OB               UInt
   // 
   //  Initial_Call         Indicates the first call of the block           Bool
   //                 1 = First call (in the case of OB1 this
   //                        is the first cycle of the CPU) 
   // 
   //  Remanence         Indicates the block is using retentive data        Bool
   //                 1 = Retentive storage has been allocated
   //                        to the block
   //  ――――――――――――――――――――――――――――――――――――――――――
   // 
   // 
   //  SI_StartUp (System Data Type)
   //  ――――――――――――――――――――――――――――――――――――――――――
   //  SIGNAL NAME          FUNCTION                     TYPE
   //  ――――――――――――――――――――――――――――――――――――――――――
   //  SI_Format          Start information format, indicates if the         USInt
   //               current OB is using block optimisation
   //                 16#FF = No information
   //                 16#FE = Block optimised
   // 
   //  OB_Class           Class  of the calling OB, for this data structure     USInt 
   //               the result is always 1 (indicating cyclic OB)
   // 
   //  OB_Nr           Number of the calling OB               UInt
   // 
   //  LostRetentive         Retentive data has been lost           Bool
   //                 1 = data has been lost
   // 
   //  LostRTC           RTC data has been lost                Bool
   //                 1 = data has been lost
   //  ――――――――――――――――――――――――――――――――――――――――――
   // 
   // 
   //                ━━━   ⬙⬙⬙⬙⬙⬙   ━━━
   // 
   // 
   // 
   // ▄▄▄▄▄▄▄▄▄▄▄▄▄▄▄▄▄▄▄▄▄▄▄▄▄▄▄▄▄▄▄▄▄▄▄▄▄▄▄▄▄▄▄▄
   // 10.     SPECIAL PROPERTIES AND REQUIREMENTS
   // 
   // 
   // 
   // ▂▂▂▂▂▂▂▂▂▂▂▂▂▂▂▂▂▂▂▂▂▂▂▂▂▂▂▂▂▂▂▂▂▂▂▂▂▂▂▂▂▂▂▂
   // 10.1   Block optimisation
   // 
   // 
   //      Block optimisation is ACTIVE for this block
   // 
   // 
   // 
   // ▂▂▂▂▂▂▂▂▂▂▂▂▂▂▂▂▂▂▂▂▂▂▂▂▂▂▂▂▂▂▂▂▂▂▂▂▂▂▂▂▂▂▂▂
   // 10.2   Calling requirements
   // 
   // 
   // This block must be the first non-debug block call within the main organisation block (OB 1). 
   // It should be in Network 3 of OB1.
   // 
   //                ━━━   ⬙⬙⬙⬙⬙⬙   ━━━
   // 
   // 
   // 
   // ▄▄▄▄▄▄▄▄▄▄▄▄▄▄▄▄▄▄▄▄▄▄▄▄▄▄▄▄▄▄▄▄▄▄▄▄▄▄▄▄▄▄▄▄
   // 11.     EXAMPLE USAGE
   // 
   // 
   //      OB1 NETWORK 3
   // 
   //                       ┌────────────
   //    ───────────────────┤ FC01001 
   //                       ├──────────
   //                  "_ClockMem" ─┤ CLOCK_MEM
   //                       │
   //  "DB21001_DY_StdGlobalData".SysSignals ─┤ SYS_SIGNALS
   //                       │
   //       "DB21001_DY_StdGlobalData".SysData ─┤ SYS_DATA
   //                       │               │
   //                       │               │
   //                              SYS_SIGNAL_TAGS├─ "_SysSignals"
   //                                    │
   //                       ─────────────┘
   // 
   // 
   //                ━━━   ⬙⬙⬙⬙⬙⬙   ━━━
   // 
   // 
   // ██████████████ █ █ █ █  END   █ █ █ █ ██████████████
END_REGION

REGION Network 3: Current revision and modification history
   // ▄▄▄▄▄▄▄▄▄▄▄▄▄▄▄▄▄▄▄▄▄▄▄▄▄▄▄▄▄▄▄▄▄▄▄▄▄▄▄▄▄▄▄▄
   // MODIFICATION HISTORY
   // 
   // 
   // The revision data shown here, in the network comments, contains additional information 
   // reflecting the software development workflow under the version control system (VCS) employed 
   // to track all software changes.
   // 
   // The VCS in use is the Git Source Code Management system in conjunction with the GitHub online 
   // hosting system. The software in its entirety is available in the GitHub remote repository:
   // 
   //      https://github.com/practicalseries/PS2001-pal-software
   // 
   // The repository is public and can be freely copied (forked in GitHub terminology) and used 
   // under the MIT licence. 
   // 
   // The MIT licence is reproduced in full in the last network of this software module.
   // 
   // 
   //  ―――――――――――――――――――――――――――――――――――――――――――
   //  DATE       REVISION             MASTER BRANCH     DEV
   //          (nnn.amm)   COMMIT TAG    (Base ---> Merge)    BRANCH   Author
   //  ———————————————————————————————————————————
   //  2021.05.11    000.801   D0005A-000.801   D0005 N/A     D0005A   M. Gledhill
   //                        FC01001 — Released for SMT
   // 
   //  2021.05.08    000.101   D0005A-000.101   D0005 N/A     D0005A   M. Gledhill
   //                        FC01001 Migration to VCS
   //  ———————————————————————————————————————————
   //   Where: nnn  =  Major revision
   //         a  =  Type (1-7 Development, 8 Proving, 9 Qualification, 0 Release)
   //       mm  =  Minor revision (must be 00 if a = 0)
   //         Block properties version number should be set to nn.a (only one decimal place)
   // 
   // ▄▄▄▄▄▄▄▄▄▄▄▄▄▄▄▄▄▄▄▄▄▄▄▄▄▄▄▄▄▄▄▄▄▄▄▄▄▄▄▄▄▄▄▄
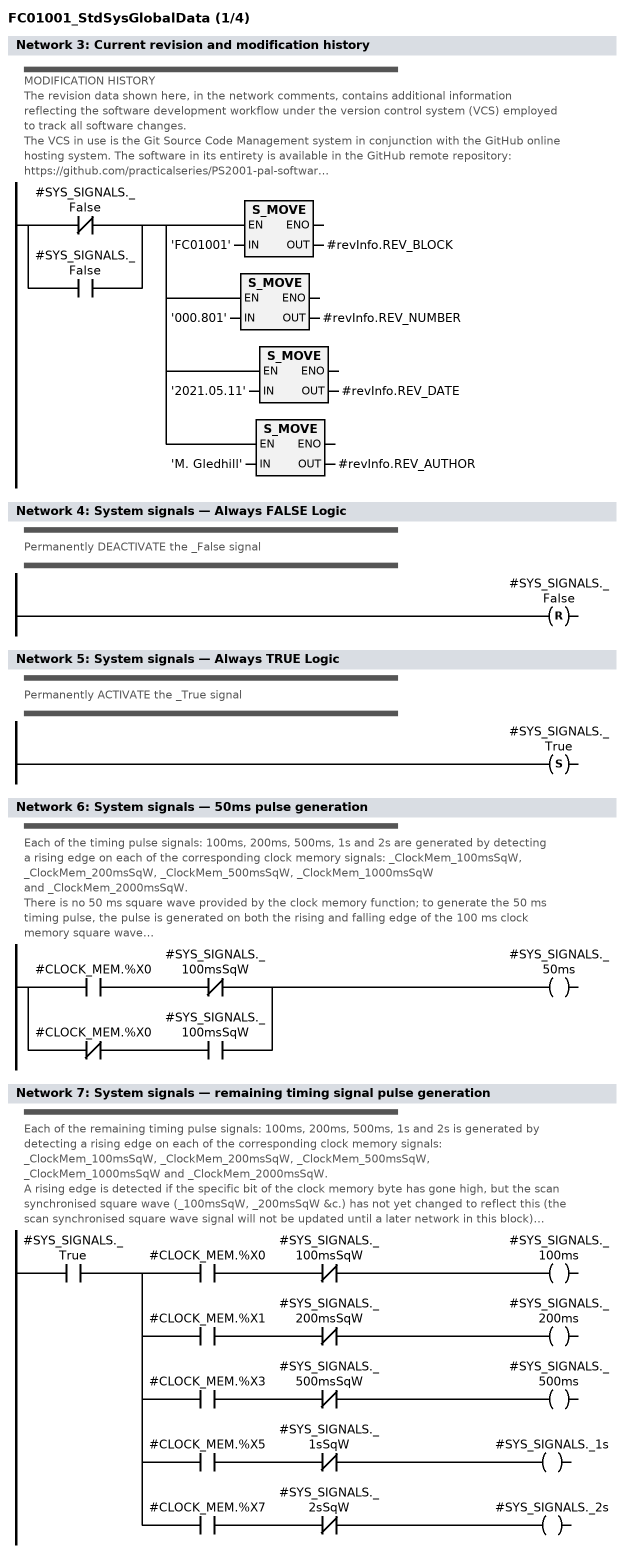
   RUNG wire#powerrail
      I_Contact( #SYS_SIGNALS._False )
      wire#w1
      S_Move(in := 'FC01001', out => #revInfo.REV_BLOCK)
   END_RUNG
   RUNG wire#powerrail
      Contact( #SYS_SIGNALS._False )
   END_RUNG wire#w1
   RUNG wire#w1
      S_Move(in := '000.801', out => #revInfo.REV_NUMBER)
   END_RUNG
   RUNG wire#w1
      S_Move(in := '2021.05.11', out => #revInfo.REV_DATE)
   END_RUNG
   RUNG wire#w1
      S_Move(in := 'M. Gledhill', out => #revInfo.REV_AUTHOR)
   END_RUNG
   // the same network as SCL:
   IF NOT #SYS_SIGNALS._False OR #SYS_SIGNALS._False THEN
       #revInfo.REV_BLOCK := 'FC01001';
       #revInfo.REV_NUMBER := '000.801';
       #revInfo.REV_DATE := '2021.05.11';
       #revInfo.REV_AUTHOR := 'M. Gledhill';
   END_IF;
END_REGION

REGION Network 4: System signals — Always FALSE Logic
   // ▀▀▀▀▀▀▀▀▀▀▀▀▀▀▀▀▀▀▀▀▀▀▀▀▀▀▀▀▀▀▀▀▀▀▀▀▀▀▀▀▀▀▀▀
   // Permanently DEACTIVATE the _False signal
   // ▄▄▄▄▄▄▄▄▄▄▄▄▄▄▄▄▄▄▄▄▄▄▄▄▄▄▄▄▄▄▄▄▄▄▄▄▄▄▄▄▄▄▄▄
   RUNG wire#powerrail
      R_Coil( #SYS_SIGNALS._False )
   END_RUNG
   // the same network as SCL:
   #SYS_SIGNALS._False := FALSE;
END_REGION

REGION Network 5: System signals — Always TRUE Logic
   // ▀▀▀▀▀▀▀▀▀▀▀▀▀▀▀▀▀▀▀▀▀▀▀▀▀▀▀▀▀▀▀▀▀▀▀▀▀▀▀▀▀▀▀▀
   // Permanently ACTIVATE the _True signal
   // ▄▄▄▄▄▄▄▄▄▄▄▄▄▄▄▄▄▄▄▄▄▄▄▄▄▄▄▄▄▄▄▄▄▄▄▄▄▄▄▄▄▄▄▄
   RUNG wire#powerrail
      S_Coil( #SYS_SIGNALS._True )
   END_RUNG
   // the same network as SCL:
   #SYS_SIGNALS._True := TRUE;
END_REGION

REGION Network 6: System signals — 50ms pulse generation
   // ▀▀▀▀▀▀▀▀▀▀▀▀▀▀▀▀▀▀▀▀▀▀▀▀▀▀▀▀▀▀▀▀▀▀▀▀▀▀▀▀▀▀▀▀
   // Each of the timing pulse signals: 100ms, 200ms, 500ms, 1s and 2s are generated by detecting 
   // a rising edge on each of the corresponding clock memory signals: _ClockMem_100msSqW, 
   // _ClockMem_200msSqW, _ClockMem_500msSqW, _ClockMem_1000msSqW 
   // and _ClockMem_2000msSqW. 
   // 
   // There is no 50 ms square wave provided by the clock memory function; to generate the 50 ms 
   // timing pulse, the pulse is generated on both the rising and falling edge of the 100 ms clock 
   // memory square wave:
   // 
   // A rising edge is detected if bit 0 of the clock memory byte has gone high, but the scan
   // synchronised square wave (_100msSqW) has not yet changed to reflect this (the _100msSqW
   // signal will not be updated until a later network in this block). I.e. a rising edge has been
   // detected.
   // 
   // The falling edge is detected in much the same way, if bit 0 of the clock memory had gone low,
   // but the _100msSqW is still high (has not yet seen the change).
   // 
   // In either case a _50ms pulse signal is generated, this is active for just one cycle.
   // ▄▄▄▄▄▄▄▄▄▄▄▄▄▄▄▄▄▄▄▄▄▄▄▄▄▄▄▄▄▄▄▄▄▄▄▄▄▄▄▄▄▄▄▄
   RUNG wire#powerrail
      Contact( #CLOCK_MEM.%X0 )
      I_Contact( #SYS_SIGNALS._100msSqW )
      wire#w1
      Coil( #SYS_SIGNALS._50ms )
   END_RUNG
   RUNG wire#powerrail
      I_Contact( #CLOCK_MEM.%X0 )
      Contact( #SYS_SIGNALS._100msSqW )
   END_RUNG wire#w1
   // the same network as SCL:
   #SYS_SIGNALS._50ms := (#CLOCK_MEM.%X0 AND NOT #SYS_SIGNALS._100msSqW) OR (NOT #CLOCK_MEM.%X0 AND #SYS_SIGNALS._100msSqW);
END_REGION

REGION Network 7: System signals — remaining timing signal pulse generation
   // ▀▀▀▀▀▀▀▀▀▀▀▀▀▀▀▀▀▀▀▀▀▀▀▀▀▀▀▀▀▀▀▀▀▀▀▀▀▀▀▀▀▀▀▀
   // Each of the remaining timing pulse signals: 100ms, 200ms, 500ms, 1s and 2s is generated by 
   // detecting a rising edge on each of the corresponding clock memory signals: 
   // _ClockMem_100msSqW, _ClockMem_200msSqW, _ClockMem_500msSqW, 
   // _ClockMem_1000msSqW and _ClockMem_2000msSqW. 
   // 
   // A rising edge is detected if the specific bit of the clock memory byte has gone high, but the scan
   // synchronised square wave (_100msSqW, _200msSqW &c.) has not yet changed to reflect this (the 
   // scan synchronised square wave signal will not be updated until a later network in this block). 
   // I.e. a rising edge has been detected.
   // 
   // The following pulses are generated:
   // 
   // 
   //  ――――――――――――――――――――――――――――――――――――――――――
   //  NAME          TYPE  DESCRIPTION
   //  ――――――――――――――――――――――――――――――――――――――――――
   //  _50ms           Bool     System Timing — 50 ms pulse 
   //  _100ms            Bool     System Timing — 100 ms pulse 
   //  _200ms            Bool     System Timing — 200 ms pulse 
   //  _500ms            Bool     System Timing — 500 ms pulse 
   //  _1s           Bool     System Timing — 1 s pulse 
   //  _2s           Bool     System Timing — 2 s pulse 
   //  ――――――――――――――――――――――――――――――――――――――――――
   // 
   // 
   // ▄▄▄▄▄▄▄▄▄▄▄▄▄▄▄▄▄▄▄▄▄▄▄▄▄▄▄▄▄▄▄▄▄▄▄▄▄▄▄▄▄▄▄▄
   RUNG wire#powerrail
      Contact( #SYS_SIGNALS._True )
      wire#w1
      Contact( #CLOCK_MEM.%X0 )
      I_Contact( #SYS_SIGNALS._100msSqW )
      Coil( #SYS_SIGNALS._100ms )
   END_RUNG
   RUNG wire#w1
      Contact( #CLOCK_MEM.%X1 )
      I_Contact( #SYS_SIGNALS._200msSqW )
      Coil( #SYS_SIGNALS._200ms )
   END_RUNG
   RUNG wire#w1
      Contact( #CLOCK_MEM.%X3 )
      I_Contact( #SYS_SIGNALS._500msSqW )
      Coil( #SYS_SIGNALS._500ms )
   END_RUNG
   RUNG wire#w1
      Contact( #CLOCK_MEM.%X5 )
      I_Contact( #SYS_SIGNALS._1sSqW )
      Coil( #SYS_SIGNALS._1s )
   END_RUNG
   RUNG wire#w1
      Contact( #CLOCK_MEM.%X7 )
      I_Contact( #SYS_SIGNALS._2sSqW )
      Coil( #SYS_SIGNALS._2s )
   END_RUNG
   // the same network as SCL:
   #SYS_SIGNALS._100ms := #SYS_SIGNALS._True AND #CLOCK_MEM.%X0 AND NOT #SYS_SIGNALS._100msSqW;
   #SYS_SIGNALS._200ms := #SYS_SIGNALS._True AND #CLOCK_MEM.%X1 AND NOT #SYS_SIGNALS._200msSqW;
   #SYS_SIGNALS._500ms := #SYS_SIGNALS._True AND #CLOCK_MEM.%X3 AND NOT #SYS_SIGNALS._500msSqW;
   #SYS_SIGNALS._1s := #SYS_SIGNALS._True AND #CLOCK_MEM.%X5 AND NOT #SYS_SIGNALS._1sSqW;
   #SYS_SIGNALS._2s := #SYS_SIGNALS._True AND #CLOCK_MEM.%X7 AND NOT #SYS_SIGNALS._2sSqW;
END_REGION

REGION Network 8: System signals — synchronised square wave generation
   // ▀▀▀▀▀▀▀▀▀▀▀▀▀▀▀▀▀▀▀▀▀▀▀▀▀▀▀▀▀▀▀▀▀▀▀▀▀▀▀▀▀▀▀▀
   // The CLOCK_MEM parameter is "sliced" into individual bits and these are passed to the scan
   // synchronised square wave global data signals (only five are used).
   // 
   // 
   //  ――――――――――――――――――――――――――――――――――――――――――
   //  CLOCK_MEM ADDRESS    BIT    DESCRIPTION
   //  ――――――――――――――――――――――――――――――――――――――――――
   //  #CLOCK_MEM.%X0    Bit 0    Clock Memory — 10.0 Hz square wave -   100ms period
   //  #CLOCK_MEM.%X1    Bit 1    Clock Memory — 5.00 Hz square wave -   200ms period
   //  #CLOCK_MEM.%X2    Bit 2    Clock Memory — 2.50 Hz square wave -   400ms period
   //  #CLOCK_MEM.%X3    Bit 3    Clock Memory — 2.00 Hz square wave -   500ms period
   //  #CLOCK_MEM.%X4    Bit 4    Clock Memory — 1.25 Hz square wave -   800ms period
   //  #CLOCK_MEM.%X5    Bit 5    Clock Memory — 1.00 Hz square wave - 1000ms period
   //  #CLOCK_MEM.%X6    Bit 6    Clock Memory — 0.62 Hz square wave - 1600ms period
   //  #CLOCK_MEM.%X7    Bit 7    Clock Memory — 0.50 Hz square wave - 2000ms period
   //  ――――――――――――――――――――――――――――――――――――――――――
   // 
   // 
   // The five signal generate the following square waves:
   // 
   // 
   //  ――――――――――――――――――――――――――――――――――――――――――
   //  NAME          TYPE  DESCRIPTION
   //  ――――――――――――――――――――――――――――――――――――――――――
   //  _100msSqW       Bool     System Timing — 100 ms square wave 
   //  _200msSqW       Bool     System Timing — 200 ms square wave 
   //  _500msSqW       Bool     System Timing — 500 ms square wave 
   //  _1sSqW            Bool     System Timing — 1 s square wave 
   //  _2sSqW            Bool     System Timing — 2 s square wave 
   //  ――――――――――――――――――――――――――――――――――――――――――
   // 
   // 
   // ▄▄▄▄▄▄▄▄▄▄▄▄▄▄▄▄▄▄▄▄▄▄▄▄▄▄▄▄▄▄▄▄▄▄▄▄▄▄▄▄▄▄▄▄
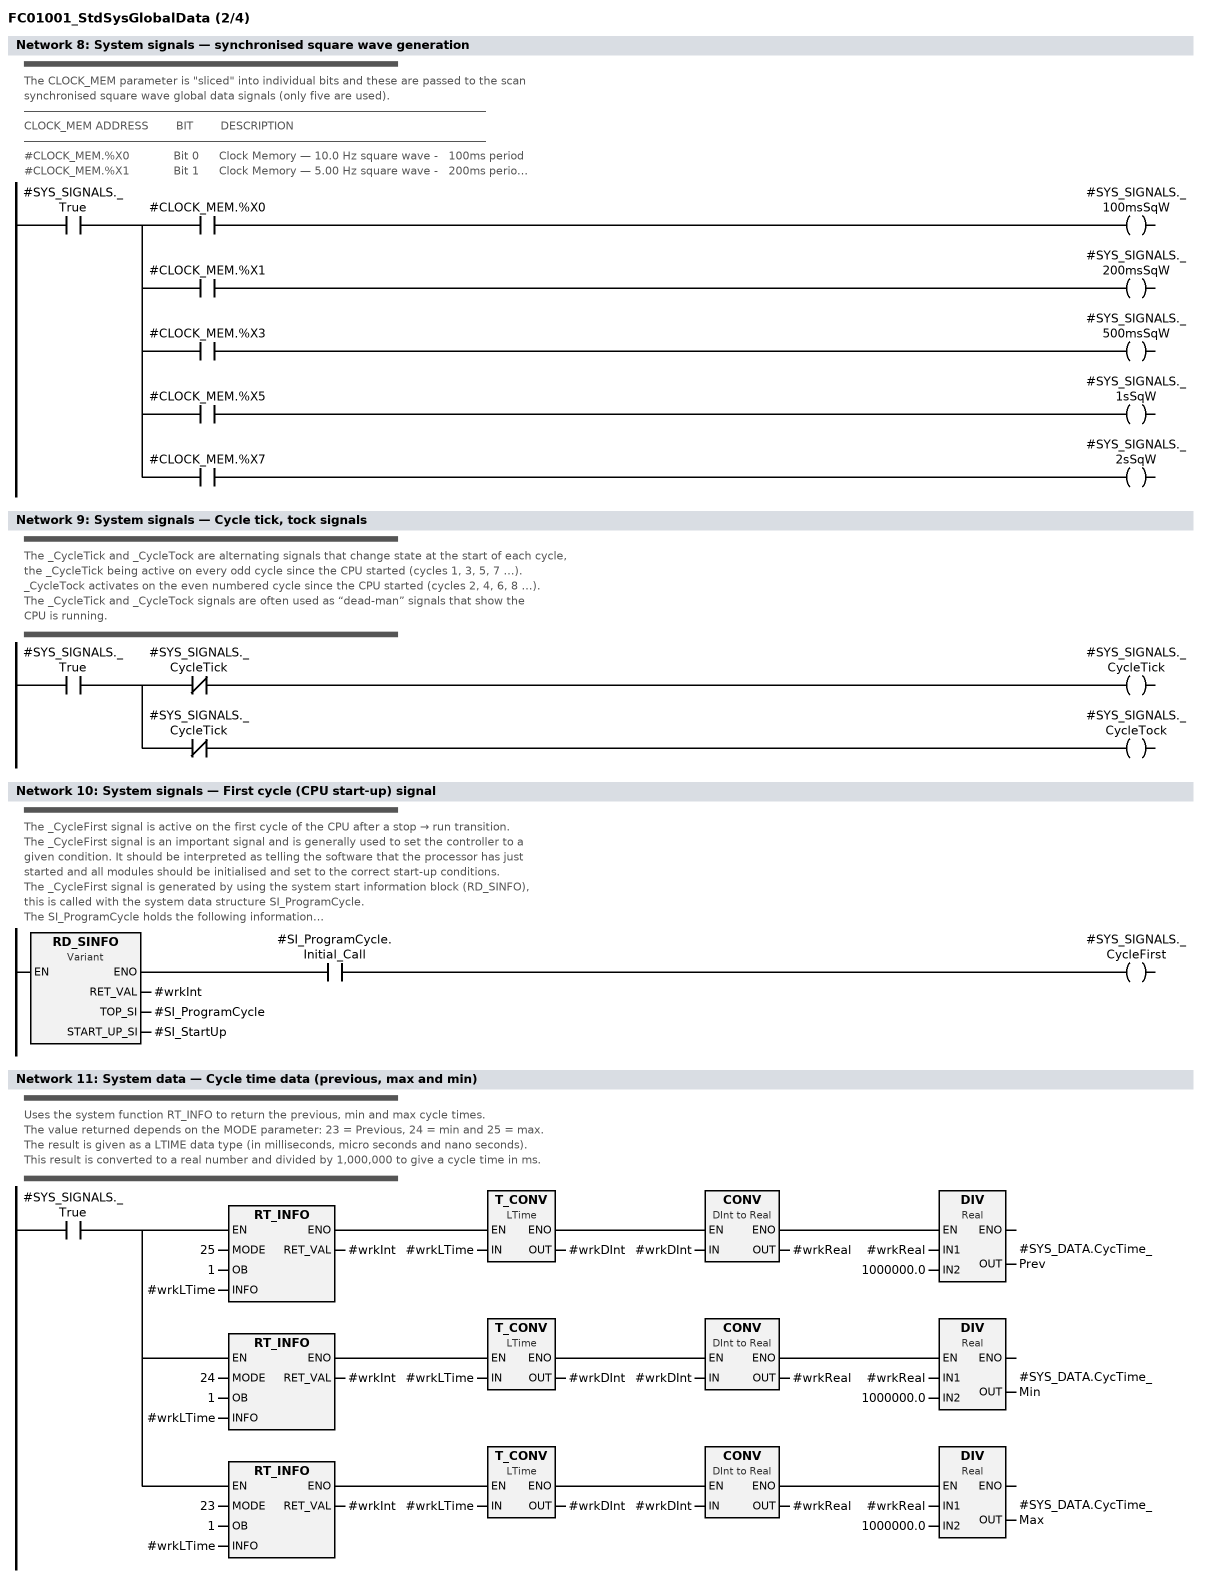
   RUNG wire#powerrail
      Contact( #SYS_SIGNALS._True )
      wire#w1
      Contact( #CLOCK_MEM.%X0 )
      Coil( #SYS_SIGNALS._100msSqW )
   END_RUNG
   RUNG wire#w1
      Contact( #CLOCK_MEM.%X1 )
      Coil( #SYS_SIGNALS._200msSqW )
   END_RUNG
   RUNG wire#w1
      Contact( #CLOCK_MEM.%X3 )
      Coil( #SYS_SIGNALS._500msSqW )
   END_RUNG
   RUNG wire#w1
      Contact( #CLOCK_MEM.%X5 )
      Coil( #SYS_SIGNALS._1sSqW )
   END_RUNG
   RUNG wire#w1
      Contact( #CLOCK_MEM.%X7 )
      Coil( #SYS_SIGNALS._2sSqW )
   END_RUNG
   // the same network as SCL:
   #SYS_SIGNALS._100msSqW := #SYS_SIGNALS._True AND #CLOCK_MEM.%X0;
   #SYS_SIGNALS._200msSqW := #SYS_SIGNALS._True AND #CLOCK_MEM.%X1;
   #SYS_SIGNALS._500msSqW := #SYS_SIGNALS._True AND #CLOCK_MEM.%X3;
   #SYS_SIGNALS._1sSqW := #SYS_SIGNALS._True AND #CLOCK_MEM.%X5;
   #SYS_SIGNALS._2sSqW := #SYS_SIGNALS._True AND #CLOCK_MEM.%X7;
END_REGION

REGION Network 9: System signals — Cycle tick, tock signals
   // ▀▀▀▀▀▀▀▀▀▀▀▀▀▀▀▀▀▀▀▀▀▀▀▀▀▀▀▀▀▀▀▀▀▀▀▀▀▀▀▀▀▀▀▀
   // The _CycleTick and _CycleTock are alternating signals that change state at the start of each cycle, 
   // the _CycleTick being active on every odd cycle since the CPU started (cycles 1, 3, 5, 7 …).
   // 
   // _CycleTock activates on the even numbered cycle since the CPU started (cycles 2, 4, 6, 8 …).
   // 
   // The _CycleTick and _CycleTock signals are often used as “dead-man” signals that show the 
   // CPU is running.
   // ▄▄▄▄▄▄▄▄▄▄▄▄▄▄▄▄▄▄▄▄▄▄▄▄▄▄▄▄▄▄▄▄▄▄▄▄▄▄▄▄▄▄▄▄
   RUNG wire#powerrail
      Contact( #SYS_SIGNALS._True )
      wire#w1
      I_Contact( #SYS_SIGNALS._CycleTick )
      Coil( #SYS_SIGNALS._CycleTick )
   END_RUNG
   RUNG wire#w1
      I_Contact( #SYS_SIGNALS._CycleTick )
      Coil( #SYS_SIGNALS._CycleTock )
   END_RUNG
   // the same network as SCL:
   #SYS_SIGNALS._CycleTick := #SYS_SIGNALS._True AND NOT #SYS_SIGNALS._CycleTick;
   #SYS_SIGNALS._CycleTock := #SYS_SIGNALS._True AND NOT #SYS_SIGNALS._CycleTick;
END_REGION

REGION Network 10: System signals — First cycle (CPU start-up) signal
   // ▀▀▀▀▀▀▀▀▀▀▀▀▀▀▀▀▀▀▀▀▀▀▀▀▀▀▀▀▀▀▀▀▀▀▀▀▀▀▀▀▀▀▀▀
   // The _CycleFirst signal is active on the first cycle of the CPU after a stop → run transition.
   // 
   // The _CycleFirst signal is an important signal and is generally used to set the controller to a 
   // given condition. It should be interpreted as telling the software that the processor has just 
   // started and all modules should be initialised and set to the correct start-up conditions.
   // 
   // The _CycleFirst signal is generated by using the system start information block (RD_SINFO), 
   // this is called with the system data structure SI_ProgramCycle.
   // 
   // The SI_ProgramCycle holds the following information:
   // 
   // 
   //  SI_ProgramCycle (System Data Type)
   //  ――――――――――――――――――――――――――――――――――――――――――
   //  SIGNAL NAME          FUNCTION                     TYPE
   //  ――――――――――――――――――――――――――――――――――――――――――
   //  SI_Format          Start information format, indicates if the         USInt
   //               current OB is using block optimisation
   //                 16#FF = No information
   //                 16#FE = Block optimised
   // 
   //  OB_Class           Class  of the calling OB, for this data structure     USInt 
   //               the result is always 1 (indicating cyclic OB)
   // 
   //  OB_Nr           Number of the calling OB               UInt
   // 
   //  Initial_Call         Indicates the first call of the block           Bool
   //                 1 = First call (in the case of OB1 this
   //                        is the first cycle of the CPU) 
   // 
   //  Remanence         Indicates the block is using retentive data        Bool
   //                 1 = Retentive storage has been allocated
   //                        to the block
   //  ――――――――――――――――――――――――――――――――――――――――――
   // 
   // 
   // If the Initial_Call signal is active, the CPU is executing the first cycle of OB 1.
   // ▄▄▄▄▄▄▄▄▄▄▄▄▄▄▄▄▄▄▄▄▄▄▄▄▄▄▄▄▄▄▄▄▄▄▄▄▄▄▄▄▄▄▄▄
   RUNG wire#powerrail
      { S7_Templates := "si_type := Variant" } RD_SINFO(RET_VAL => #wrkInt, TOP_SI => #SI_ProgramCycle, START_UP_SI => #SI_StartUp)
      Contact( #SI_ProgramCycle.Initial_Call )
      Coil( #SYS_SIGNALS._CycleFirst )
   END_RUNG
   // the same network as SCL:
   #wrkInt := RD_SINFO(TOP_SI => #SI_ProgramCycle, START_UP_SI => #SI_StartUp, ENO => #_w1);
   #SYS_SIGNALS._CycleFirst := #_w1 AND #SI_ProgramCycle.Initial_Call;
END_REGION

REGION Network 11: System data — Cycle time data (previous, max and min)
   // ▀▀▀▀▀▀▀▀▀▀▀▀▀▀▀▀▀▀▀▀▀▀▀▀▀▀▀▀▀▀▀▀▀▀▀▀▀▀▀▀▀▀▀▀
   // Uses the system function RT_INFO to return the previous, min and max cycle times. 
   // 
   // The value returned depends on the MODE parameter: 23 = Previous, 24 = min and 25 = max.
   // 
   // The result is given as a LTIME data type (in milliseconds, micro seconds and nano seconds). 
   // This result is converted to a real number and divided by 1,000,000 to give a cycle time in ms.
   // ▄▄▄▄▄▄▄▄▄▄▄▄▄▄▄▄▄▄▄▄▄▄▄▄▄▄▄▄▄▄▄▄▄▄▄▄▄▄▄▄▄▄▄▄
   RUNG wire#powerrail
      Contact( #SYS_SIGNALS._True )
      wire#w1
      RT_INFO(MODE := 25, OB := 1, INFO := #wrkLTime, Ret_Val => #wrkInt)
      { S7_Templates := "[src_type := LTime, dest_type := DInt]" } T_CONV(IN := #wrkLTime, OUT => #wrkDInt)
      { S7_Templates := "[SrcType := DInt, DestType := Real]" } Convert(in := #wrkDInt, out => #wrkReal)
      { S7_Templates := "SrcType := Real" } Div(in1 := #wrkReal, in2 := 1000000.0, out => #SYS_DATA.CycTime_Prev)
   END_RUNG
   RUNG wire#w1
      RT_INFO(MODE := 24, OB := 1, INFO := #wrkLTime, Ret_Val => #wrkInt)
      { S7_Templates := "[src_type := LTime, dest_type := DInt]" } T_CONV(IN := #wrkLTime, OUT => #wrkDInt)
      { S7_Templates := "[SrcType := DInt, DestType := Real]" } Convert(in := #wrkDInt, out => #wrkReal)
      { S7_Templates := "SrcType := Real" } Div(in1 := #wrkReal, in2 := 1000000.0, out => #SYS_DATA.CycTime_Min)
   END_RUNG
   RUNG wire#w1
      RT_INFO(MODE := 23, OB := 1, INFO := #wrkLTime, Ret_Val => #wrkInt)
      { S7_Templates := "[src_type := LTime, dest_type := DInt]" } T_CONV(IN := #wrkLTime, OUT => #wrkDInt)
      { S7_Templates := "[SrcType := DInt, DestType := Real]" } Convert(in := #wrkDInt, out => #wrkReal)
      { S7_Templates := "SrcType := Real" } Div(in1 := #wrkReal, in2 := 1000000.0, out => #SYS_DATA.CycTime_Max)
   END_RUNG
   // the same network as SCL:
   #wrkInt := RT_INFO(EN := #SYS_SIGNALS._True, MODE := 25, OB := 1, INFO := #wrkLTime, ENO => #_w1);
   T_CONV(EN := #_w1, IN := #wrkLTime, OUT => #wrkDInt, ENO => #_w2);
   IF #_w2 THEN
       #wrkReal := DINT_TO_REAL(#wrkDInt);
       #SYS_DATA.CycTime_Prev := #wrkReal / 1000000.0;
   END_IF;
   #wrkInt := RT_INFO(EN := #SYS_SIGNALS._True, MODE := 24, OB := 1, INFO := #wrkLTime, ENO => #_w3);
   T_CONV(EN := #_w3, IN := #wrkLTime, OUT => #wrkDInt, ENO => #_w4);
   IF #_w4 THEN
       #wrkReal := DINT_TO_REAL(#wrkDInt);
       #SYS_DATA.CycTime_Min := #wrkReal / 1000000.0;
   END_IF;
   #wrkInt := RT_INFO(EN := #SYS_SIGNALS._True, MODE := 23, OB := 1, INFO := #wrkLTime, ENO => #_w5);
   T_CONV(EN := #_w5, IN := #wrkLTime, OUT => #wrkDInt, ENO => #_w6);
   IF #_w6 THEN
       #wrkReal := DINT_TO_REAL(#wrkDInt);
       #SYS_DATA.CycTime_Max := #wrkReal / 1000000.0;
   END_IF;
END_REGION

REGION Network 12: System data — Cycle counter
   // ▀▀▀▀▀▀▀▀▀▀▀▀▀▀▀▀▀▀▀▀▀▀▀▀▀▀▀▀▀▀▀▀▀▀▀▀▀▀▀▀▀▀▀▀
   // The Cyc_Counter signal is simply an unsigned double integer (UDint) that is incremented by one 
   // each scan. The counter can count up to 4.3 billion cycles (4,294,967,296) before repeating (at an 
   // average cycle time of 15 ms, it would be two years before the counter wrapped around and 
   // started again at zero).
   // 
   // The Cyc_Counter signal is reset to zero if the CPU is restarted (_CycleFirst signal is triggered), it is 
   // also reset to zero if the count exceeds the maximum value for a UDint (4,294,967,296).
   // ▄▄▄▄▄▄▄▄▄▄▄▄▄▄▄▄▄▄▄▄▄▄▄▄▄▄▄▄▄▄▄▄▄▄▄▄▄▄▄▄▄▄▄▄
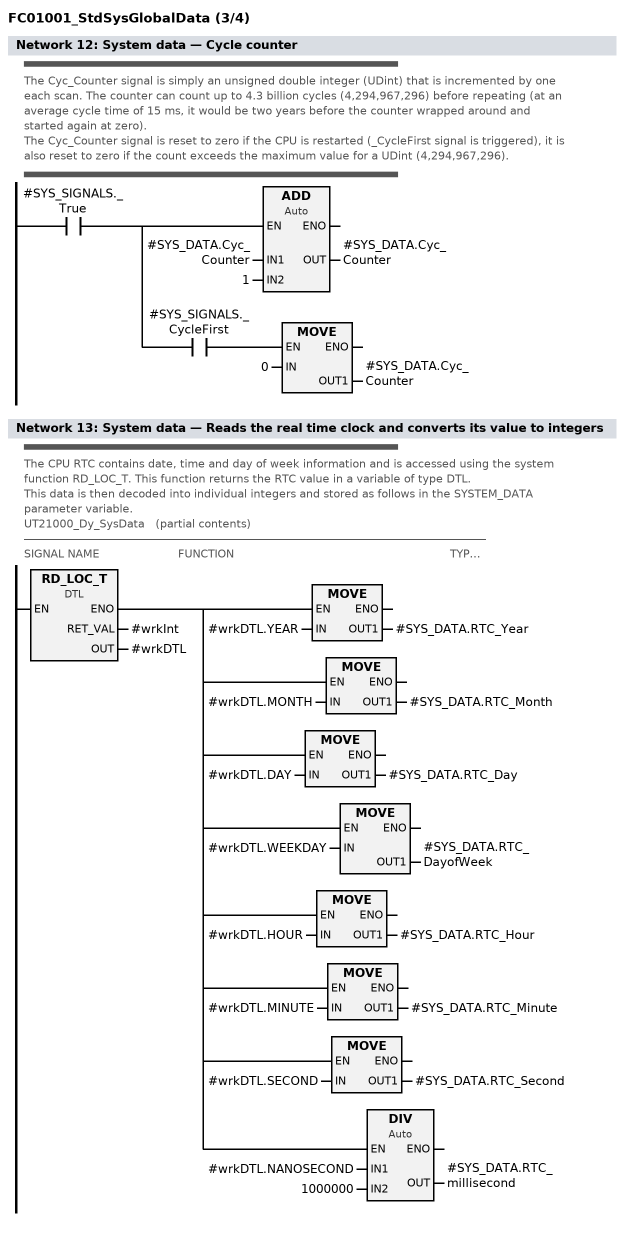
   RUNG wire#powerrail
      Contact( #SYS_SIGNALS._True )
      wire#w1
      { S7_GenerateENO := "TRUE" } Add(in1 := #SYS_DATA.Cyc_Counter, in2 := 1, out => #SYS_DATA.Cyc_Counter)
   END_RUNG
   RUNG wire#w1
      Contact( #SYS_SIGNALS._CycleFirst )
      Move(in := 0, out1 => #SYS_DATA.Cyc_Counter)
   END_RUNG
   // the same network as SCL:
   IF #SYS_SIGNALS._True THEN #SYS_DATA.Cyc_Counter := #SYS_DATA.Cyc_Counter + 1; END_IF;
   IF #SYS_SIGNALS._True AND #SYS_SIGNALS._CycleFirst THEN #SYS_DATA.Cyc_Counter := 0; END_IF;
END_REGION

REGION Network 13: System data — Reads the real time clock and converts its value to integers
   // ▀▀▀▀▀▀▀▀▀▀▀▀▀▀▀▀▀▀▀▀▀▀▀▀▀▀▀▀▀▀▀▀▀▀▀▀▀▀▀▀▀▀▀▀
   // The CPU RTC contains date, time and day of week information and is accessed using the system 
   // function RD_LOC_T. This function returns the RTC value in a variable of type DTL.
   // 
   // This data is then decoded into individual integers and stored as follows in the SYSTEM_DATA
   // parameter variable.
   // 
   // 
   //  UT21000_Dy_SysData (partial contents)
   //  ――――――――――――――――――――――――――――――――――――――――――
   //  SIGNAL NAME          FUNCTION                     TYPE
   //  ――――――――――――――――――――――――――――――――――――――――――
   //  RTC_Year            Year (returns a value in the range 1970 to 2262)     UInt
   //  RTC_Month         Month (1-12 representing Jan to Dec)        UInt
   //  RTC_Day          Day of month (1-31)                  UInt
   //  RTC_DayOfWeek         Day of week (1-7, where 1=Sunday, 7=Saturday)    UInt
   //  RTC_Hour           Hour of day (0-23)                UInt
   //  RTC_Minute           Minutes (0-59)                   UInt
   //  RTC_Second         Seconds (0-59)                  UInt
   //  RTC_Millisecond         Milliseconds (0-999)                  UInt
   //  ――――――――――――――――――――――――――――――――――――――――――
   // 
   // 
   // The RD_LOC_T returns a nanosecond value from the RTC, this is divided by 1,000,000 to convert it 
   // to milliseconds.
   // 
   // Note:    The RTC data is local to the time zone set in the CPU and adopts any local daylight 
   //      saving that is in effect.
   // ▄▄▄▄▄▄▄▄▄▄▄▄▄▄▄▄▄▄▄▄▄▄▄▄▄▄▄▄▄▄▄▄▄▄▄▄▄▄▄▄▄▄▄▄
   RUNG wire#powerrail
      { S7_Templates := "date_type := DTL" } RD_LOC_T(RET_VAL => #wrkInt, OUT => #wrkDTL)
      wire#w1
      Move(in := #wrkDTL.YEAR, out1 => #SYS_DATA.RTC_Year)
   END_RUNG
   RUNG wire#w1
      Move(in := #wrkDTL.MONTH, out1 => #SYS_DATA.RTC_Month)
   END_RUNG
   RUNG wire#w1
      Move(in := #wrkDTL.DAY, out1 => #SYS_DATA.RTC_Day)
   END_RUNG
   RUNG wire#w1
      Move(in := #wrkDTL.WEEKDAY, out1 => #SYS_DATA.RTC_DayofWeek)
   END_RUNG
   RUNG wire#w1
      Move(in := #wrkDTL.HOUR, out1 => #SYS_DATA.RTC_Hour)
   END_RUNG
   RUNG wire#w1
      Move(in := #wrkDTL.MINUTE, out1 => #SYS_DATA.RTC_Minute)
   END_RUNG
   RUNG wire#w1
      Move(in := #wrkDTL.SECOND, out1 => #SYS_DATA.RTC_Second)
   END_RUNG
   RUNG wire#w1
      Div(in1 := #wrkDTL.NANOSECOND, in2 := 1000000, out => #SYS_DATA.RTC_millisecond)
   END_RUNG
   // the same network as SCL:
   #wrkInt := RD_LOC_T(OUT => #wrkDTL, ENO => #_w1);
   IF #_w1 THEN
       #SYS_DATA.RTC_Year := #wrkDTL.YEAR;
       #SYS_DATA.RTC_Month := #wrkDTL.MONTH;
       #SYS_DATA.RTC_Day := #wrkDTL.DAY;
       #SYS_DATA.RTC_DayofWeek := #wrkDTL.WEEKDAY;
       #SYS_DATA.RTC_Hour := #wrkDTL.HOUR;
       #SYS_DATA.RTC_Minute := #wrkDTL.MINUTE;
       #SYS_DATA.RTC_Second := #wrkDTL.SECOND;
       #SYS_DATA.RTC_millisecond := #wrkDTL.NANOSECOND / 1000000;
   END_IF;
END_REGION

REGION Network 14: System signals — Copy data to memory bit area
   // ▀▀▀▀▀▀▀▀▀▀▀▀▀▀▀▀▀▀▀▀▀▀▀▀▀▀▀▀▀▀▀▀▀▀▀▀▀▀▀▀▀▀▀▀
   // Copies all the system logic and timing signals to the SYS_SIGNAL_TAGS parameter.
   // ▄▄▄▄▄▄▄▄▄▄▄▄▄▄▄▄▄▄▄▄▄▄▄▄▄▄▄▄▄▄▄▄▄▄▄▄▄▄▄▄▄▄▄▄
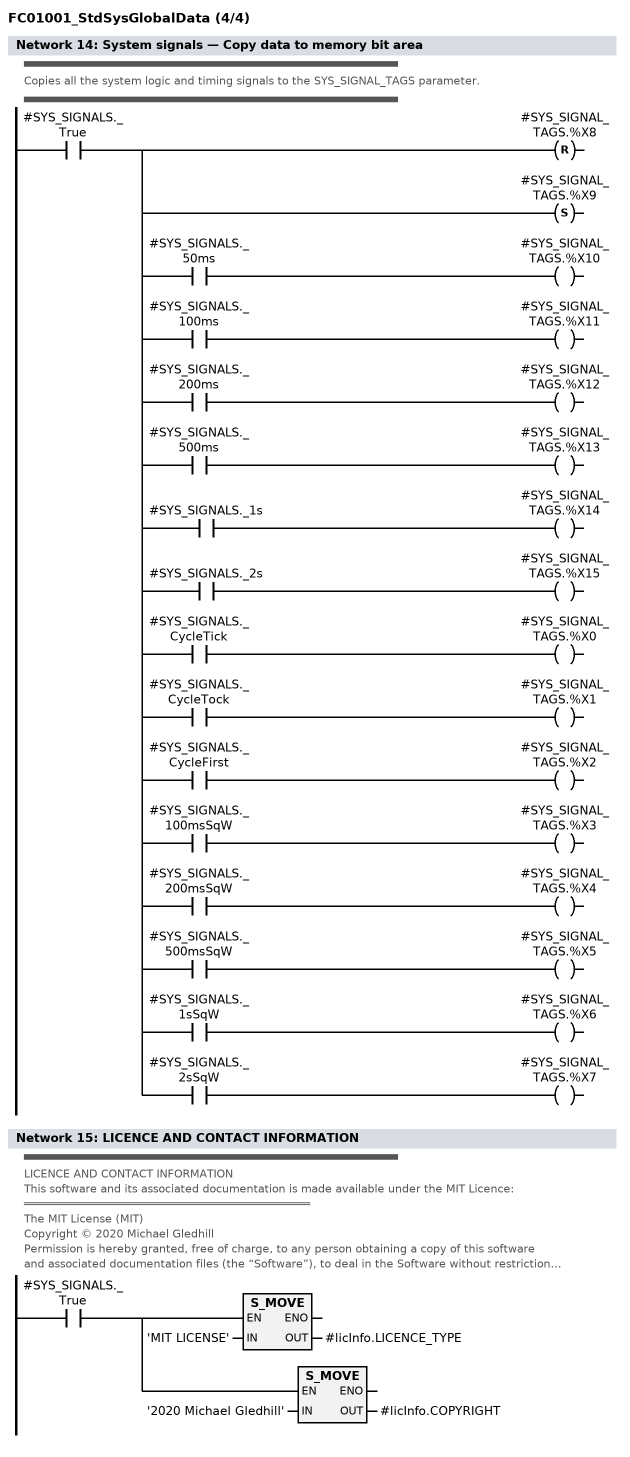
   RUNG wire#powerrail
      Contact( #SYS_SIGNALS._True )
      wire#w1
      R_Coil( #SYS_SIGNAL_TAGS.%X8 )
   END_RUNG
   RUNG wire#w1
      S_Coil( #SYS_SIGNAL_TAGS.%X9 )
   END_RUNG
   RUNG wire#w1
      Contact( #SYS_SIGNALS._50ms )
      Coil( #SYS_SIGNAL_TAGS.%X10 )
   END_RUNG
   RUNG wire#w1
      Contact( #SYS_SIGNALS._100ms )
      Coil( #SYS_SIGNAL_TAGS.%X11 )
   END_RUNG
   RUNG wire#w1
      Contact( #SYS_SIGNALS._200ms )
      Coil( #SYS_SIGNAL_TAGS.%X12 )
   END_RUNG
   RUNG wire#w1
      Contact( #SYS_SIGNALS._500ms )
      Coil( #SYS_SIGNAL_TAGS.%X13 )
   END_RUNG
   RUNG wire#w1
      Contact( #SYS_SIGNALS._1s )
      Coil( #SYS_SIGNAL_TAGS.%X14 )
   END_RUNG
   RUNG wire#w1
      Contact( #SYS_SIGNALS._2s )
      Coil( #SYS_SIGNAL_TAGS.%X15 )
   END_RUNG
   RUNG wire#w1
      Contact( #SYS_SIGNALS._CycleTick )
      Coil( #SYS_SIGNAL_TAGS.%X0 )
   END_RUNG
   RUNG wire#w1
      Contact( #SYS_SIGNALS._CycleTock )
      Coil( #SYS_SIGNAL_TAGS.%X1 )
   END_RUNG
   RUNG wire#w1
      Contact( #SYS_SIGNALS._CycleFirst )
      Coil( #SYS_SIGNAL_TAGS.%X2 )
   END_RUNG
   RUNG wire#w1
      Contact( #SYS_SIGNALS._100msSqW )
      Coil( #SYS_SIGNAL_TAGS.%X3 )
   END_RUNG
   RUNG wire#w1
      Contact( #SYS_SIGNALS._200msSqW )
      Coil( #SYS_SIGNAL_TAGS.%X4 )
   END_RUNG
   RUNG wire#w1
      Contact( #SYS_SIGNALS._500msSqW )
      Coil( #SYS_SIGNAL_TAGS.%X5 )
   END_RUNG
   RUNG wire#w1
      Contact( #SYS_SIGNALS._1sSqW )
      Coil( #SYS_SIGNAL_TAGS.%X6 )
   END_RUNG
   RUNG wire#w1
      Contact( #SYS_SIGNALS._2sSqW )
      Coil( #SYS_SIGNAL_TAGS.%X7 )
   END_RUNG
   // the same network as SCL:
   IF #SYS_SIGNALS._True THEN
       #SYS_SIGNAL_TAGS.%X8 := FALSE;
       #SYS_SIGNAL_TAGS.%X9 := TRUE;
   END_IF;
   #SYS_SIGNAL_TAGS.%X10 := #SYS_SIGNALS._True AND #SYS_SIGNALS._50ms;
   #SYS_SIGNAL_TAGS.%X11 := #SYS_SIGNALS._True AND #SYS_SIGNALS._100ms;
   #SYS_SIGNAL_TAGS.%X12 := #SYS_SIGNALS._True AND #SYS_SIGNALS._200ms;
   #SYS_SIGNAL_TAGS.%X13 := #SYS_SIGNALS._True AND #SYS_SIGNALS._500ms;
   #SYS_SIGNAL_TAGS.%X14 := #SYS_SIGNALS._True AND #SYS_SIGNALS._1s;
   #SYS_SIGNAL_TAGS.%X15 := #SYS_SIGNALS._True AND #SYS_SIGNALS._2s;
   #SYS_SIGNAL_TAGS.%X0 := #SYS_SIGNALS._True AND #SYS_SIGNALS._CycleTick;
   #SYS_SIGNAL_TAGS.%X1 := #SYS_SIGNALS._True AND #SYS_SIGNALS._CycleTock;
   #SYS_SIGNAL_TAGS.%X2 := #SYS_SIGNALS._True AND #SYS_SIGNALS._CycleFirst;
   #SYS_SIGNAL_TAGS.%X3 := #SYS_SIGNALS._True AND #SYS_SIGNALS._100msSqW;
   #SYS_SIGNAL_TAGS.%X4 := #SYS_SIGNALS._True AND #SYS_SIGNALS._200msSqW;
   #SYS_SIGNAL_TAGS.%X5 := #SYS_SIGNALS._True AND #SYS_SIGNALS._500msSqW;
   #SYS_SIGNAL_TAGS.%X6 := #SYS_SIGNALS._True AND #SYS_SIGNALS._1sSqW;
   #SYS_SIGNAL_TAGS.%X7 := #SYS_SIGNALS._True AND #SYS_SIGNALS._2sSqW;
END_REGION

REGION Network 15: LICENCE AND CONTACT INFORMATION
   // ▀▀▀▀▀▀▀▀▀▀▀▀▀▀▀▀▀▀▀▀▀▀▀▀▀▀▀▀▀▀▀▀▀▀▀▀▀▀▀▀▀▀▀▀
   // LICENCE AND CONTACT INFORMATION
   // 
   // This software and its associated documentation is made available under the MIT Licence:
   // 
   // ════════════════════════════════════════════
   // 
   // The MIT License (MIT)
   // 
   // Copyright © 2020 Michael Gledhill
   // 
   // Permission is hereby granted, free of charge, to any person obtaining a copy of this software 
   // and associated documentation files (the “Software”), to deal in the Software without restriction, 
   // including without limitation the rights to use, copy, modify, merge, publish, distribute, 
   // sublicense, and/or sell copies of the Software, and to permit persons to whom the Software is 
   // furnished to do so, subject to the following conditions: 
   // 
   // The above copyright notice and this permission notice shall be included in all copies or 
   // substantial portions of the Software.
   // 
   // THE SOFTWARE IS PROVIDED “AS IS”, WITHOUT WARRANTY OF ANY KIND, EXPRESS OR IMPLIED, 
   // INCLUDING BUT NOT LIMITED TO THE WARRANTIES OF MERCHANTABILITY, FITNESS FOR A 
   // PARTICULAR PURPOSE AND NON-INFRINGEMENT. IN NO EVENT SHALL THE AUTHORS OR COPYRIGHT 
   // HOLDERS BE LIABLE FOR ANY CLAIM, DAMAGES OR OTHER LIABILITY, WHETHER IN AN ACTION OF 
   // CONTRACT, TORT OR OTHERWISE, ARISING FROM, OUT OF OR IN CONNECTION WITH THE SOFTWARE 
   // OR THE USE OR OTHER DEALINGS IN THE SOFTWARE.
   // 
   // ════════════════════════════════════════════
   //                    ┌────────────┐
   // You can reach the author by email here:   │  mg@practicalseries.com  │
   //                    └────────────┘
   // Questions, corrections, constructive criticism and complaints (polite ones) are invited.
   // 
   // ▄▄▄▄▄▄▄▄▄▄▄▄▄▄▄▄▄▄▄▄▄▄▄▄▄▄▄▄▄▄▄▄▄▄▄▄▄▄▄▄▄▄▄▄
   RUNG wire#powerrail
      Contact( #SYS_SIGNALS._True )
      wire#w1
      S_Move(in := 'MIT LICENSE', out => #licInfo.LICENCE_TYPE)
   END_RUNG
   RUNG wire#w1
      S_Move(in := '2020 Michael Gledhill', out => #licInfo.COPYRIGHT)
   END_RUNG
   // the same network as SCL:
   IF #SYS_SIGNALS._True THEN
       #licInfo.LICENCE_TYPE := 'MIT LICENSE';
       #licInfo.COPYRIGHT := '2020 Michael Gledhill';
   END_IF;
END_REGION
END_FUNCTION

ORGANIZATION_BLOCK "OB00030_IntNCyclic_100ms"   // OB30, LAD, CyclicInterrupt
{ S7_Optimized_Access := 'TRUE' }
VERSION : 0.1
// stored: AutoNumber true, IsIECCheckEnabled false, SetENOAutomatically false
   VAR_INPUT
      Initial_Call : Bool;   // Initial call of this OB
      Event_Count : Int;   // Events discarded
   END_VAR
BEGIN

REGION Network 1: 2nd Order Response Simulation
   // ▀▀▀▀▀▀▀▀▀▀▀▀▀▀▀▀▀▀▀▀▀▀▀▀▀▀▀▀▀▀▀▀▀▀▀▀▀▀▀▀▀▀▀▀
   // Generates (in this case) a unit step response to a second order transfer function
   // ▄▄▄▄▄▄▄▄▄▄▄▄▄▄▄▄▄▄▄▄▄▄▄▄▄▄▄▄▄▄▄▄▄▄▄▄▄▄▄▄▄▄▄▄
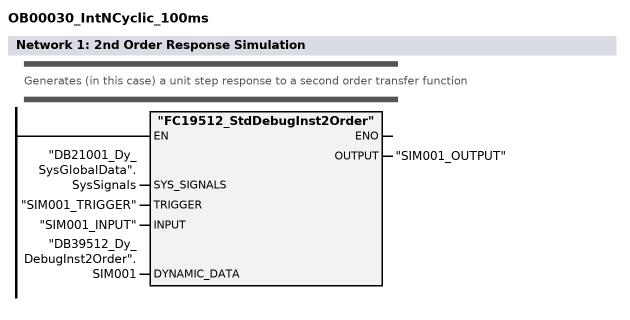
   RUNG wire#powerrail
      "FC19512_StdDebugInst2Order"(SYS_SIGNALS := "DB21001_Dy_SysGlobalData".SysSignals, TRIGGER := "SIM001_TRIGGER", INPUT := "SIM001_INPUT", DYNAMIC_DATA := "DB39512_Dy_DebugInst2Order".SIM001, OUTPUT => "SIM001_OUTPUT")
   END_RUNG
   // the same network as SCL:
   "FC19512_StdDebugInst2Order"(SYS_SIGNALS := "DB21001_Dy_SysGlobalData".SysSignals,
                           TRIGGER := "SIM001_TRIGGER",
                           INPUT := "SIM001_INPUT",
                           DYNAMIC_DATA := "DB39512_Dy_DebugInst2Order".SIM001,
                           OUTPUT => "SIM001_OUTPUT");
END_REGION
END_ORGANIZATION_BLOCK

FUNCTION "FC19512_StdDebugInst2Order" : Void   // FC19512, LAD
TITLE = Standard Module [Debug] — Second Order Response Simulation
{ S7_Optimized_Access := 'TRUE' }
AUTHOR : M_Gledhill
FAMILY : DeviceDriver
NAME : StdDebugInst2Order
VERSION : 0.1
// PRACTICAL SERIES AUTOMATION LIBRARY (PAL)   —   COPYRIGHT 2020 – M. GLEDHILL (MIT LICENCE)
//                   ———— ◆ ————
//  FOR DETAILED DOCUMENTATION — SELECT THE BLOCK IN THE PROJECT TREE AND PRESS SHIFT + F1
//  FULL ONLINE DOCUMENTATION IS AVAILABLE AT: https://practicalseries.com/2001-pal/index.html
// stored: AutoNumber false, IsIECCheckEnabled false, SetENOAutomatically false, UDAEnableTagReadback false
   VAR_INPUT
      SYS_SIGNALS : "UT21000_Dy_SysSignals";   // Common system signals — logic and timing signals
      FBK_OPEN : Bool;   // Positive open position feedback (1 = valve open, 0 = valve not open)
      FBK_CLOSED : Bool;   // Positive closed position feedback (1 = valve closed, 0 = valve not closed)
      EXT_FAULT : Bool;   // Device external fault signal (1 = fault, 0 = healthy)
      E_STOP : Bool;   // Safety (E-STOP) signal (1 = ESTOP active, 0 = healthy)
      TRIP : Bool;   // Interlock (TRIP) signal (1 = TRIP active, 0 = healthy)
      INTERLOCK : Bool;   // Interlock (INTERLOCK) signal (1 = INTERLOCK active, 0 = healthy)
      PERMISSIVE : Bool;   // Interlock (PERMISSIVE) signal (1 = PERMISSIVE active, 0 = healthy)
      STATIC_DATA : "UT11001_St_DevValveIsol";   // Static data storage (UDT)
   END_VAR
   VAR_OUTPUT
      OPERATE : Bool;   // Valve operate signal (1 = energise the valve, 0 = deenergise the valve)
   END_VAR
   VAR_IN_OUT
      DYNAMIC_DATA : "UT31001_Dy_DevValveIsol";   // Dynamic data storage (UDT)
   END_VAR
   VAR_TEMP
      revInfo : "UT01000_St_SysRevision";   // Revision information for this block
      licInfo : "UT01001_St_SysLicence";   // Licensing information for this block
      calcClosedElapsedTime : Real;   // Calculation - Derived closed signal elapsed time limit
      calcOpenElapsedTime : Real;   // Calculation - Derived open signal elapsed time limit
      wrkOpen : Bool;   // Working - open position feedback signal (actual or derived)
      wrkClosed : Bool;   // Working - closed position feedback signal (actual or derived)
      wrkCtrlPriority40 : Bool;   // Working - priority 40 condition controls the valve
      wrkCtrlPriority30 : Bool;   // Working - priority 30 condition controls the valve
      wrkCtrlPriority20 : Bool;   // Working - priority 20 condition controls the valve
      wrkCtrlPriority10 : Bool;   // Working - priority 10 condition controls the valve
      wrkCtrlPriority00 : Bool;   // Working - priority 00 condition controls the valve
      wrkCtrlAutManOpCl : Bool;   // Working - consolidated auto/manual open or close request
      wrkTimeFbkOpenSim : Real;   // Working - value of opening timer before derived open feedback
      wrkTimeFbkClosedSim : Real;   // Working - value of closing timer before derived closed feedback
      wrkInt : Int;   // Working - storage area (integer)
      wrkReal : Real;   // Working - storage (Real)
      wrkDInt : DInt;   // Working - storage area (double integer)
   END_VAR
   VAR CONSTANT
      k_TIME_OP_MIN : Real := 0.21;   // Minimum value for the valve operation timer
   END_VAR
BEGIN

